// TIA Portal V20 export
FUNCTION_BLOCK "Sequence_1_SemiAutoSplice"   // FB124, LAD
TITLE = Sequence
// Sequence template programmend in ladder logic
// stored: IsIECCheckEnabled true, MemoryReserve 100, Namespace Unit1.Em2, SetENOAutomatically true
   VAR
      instSequenceLADControl { ExternalWritable := 'False'} : "LAF_ControlLadSequence";
      instSequenceLADStatus { ExternalWritable := 'False'} : "LAF_StatusLadSequence";
      statPulse { ExternalWritable := 'False'} : Array[0..999] of Bool;
      statTonTimer { ExternalWritable := 'False'} : Array[0..9999] of TON_TIME;
   END_VAR
   VAR_TEMP
      tempCustomerAction : Bool;   // Placeholder for possible actions
      tempDo_nothing_and_wait_for_init : Bool;   // Placeholder for doing nothing
      tempSafeStateCondition : Bool;   // Temp Condition for the equipment module to be in a safe state
   END_VAR
   VAR CONSTANT
      STEP_IDLE : DInt := 1;   // Idle Step
      JOB_1_STEP_01 : DInt := 101;   // Template Step
      JOB_1_STEP_11 : DInt := 111;   // Template Step
      JOB_2_STEP_01 : DInt := 201;   // Template Step
      JOB_2_STEP_11 : DInt := 211;   // Template Step
      JOB_2_STEP_21 : DInt := 221;   // Template Step
      JOB_2_STEP_31 : DInt := 231;   // Template Step
      JOB_2_STEP_41 : DInt := 241;   // Template Step
      JOB_3_STEP_01 : DInt := 301;   // Template Step
      JOB_3_STEP_03 : DInt := 303;
      JOB_3_STEP_11 : DInt := 311;
      JOB_3_STEP_21 : DInt := 321;
      JOB_3_STEP_31 : DInt := 331;
      JOB_3_STEP_41 : DInt := 341;
      JOB_3_STEP_51 : DInt := 351;
      JOB_4_STEP_01 : DInt := 401;   // Template Step
      JOB_4_STEP_03 : DInt := 403;   // Template Step
      JOB_4_STEP_11 : DInt := 411;   // Template Step
      JOB_4_STEP_21 : DInt := 421;   // Template Step
      JOB_4_STEP_31 : DInt := 431;   // Template Step
      JOB_4_STEP_41 : DInt := 441;
      JOB_4_STEP_51 : DInt := 451;
      JOB_5_STEP_01 : DInt := 501;   // Template Step
      JOB_6_STEP_01 : DInt := 601;   // Template Step
      JOB_7_STEP_01 : DInt := 701;   // Template Step
      JOB_7_STEP_11 : DInt := 711;   // Template Step
      JOB_7_STEP_21 : DInt := 721;   // Template Step
      JOB_7_STEP_31 : DInt := 731;   // Template Step
      JOB_8_STEP_01 : DInt := 801;   // Template Step
      JOB_8_STEP_11 : DInt := 811;   // Template Step
      JOB_9_STEP_01 : DInt := 901;   // Template Step
      JOB_9_STEP_11 : DInt := 911;   // Template Step
      JOB_9_STEP_21 : DInt := 921;   // Template Step
      JOB_10_STEP_01 : DInt := 1001;   // Template Step
      JOB_10_STEP_11 : DInt := 1011;   // Template Step
      JOB_10_STEP_21 : DInt := 1021;   // Template Step
      JOB_10_STEP_31 : DInt := 1031;   // Template Step
      JOB_10_STEP_41 : DInt := 1041;   // Template Step
      JOB_11_STEP_01 : DInt := 1101;   // Template Step
      JOB_11_STEP_11 : DInt := 1111;   // Template Step
      JOB_11_STEP_21 : DInt := 1121;   // Template Step
      JOB_12_STEP_01 : DInt := 1201;   // Template Step
      JOB_12_STEP_11 : DInt := 1211;   // Template Step
      JOB_12_STEP_21 : DInt := 1221;   // Template Step
      JOB_13_STEP_01 : DInt := 1301;   // Template Step
      JOB_13_STEP_11 : DInt := 1311;   // Template Step
      JOB_13_STEP_21 : DInt := 1321;   // Template Step
      JOB_13_STEP_31 : DInt := 1331;   // Template Step
      JOB_13_STEP_41 : DInt := 1341;   // Template Step
      JOB_13_STEP_45 : DInt := 1345;   // Template Step
      JOB_13_STEP_46 : DInt := 1346;   // Template Step
      JOB_13_STEP_48 : DInt := 1348;   // Template Step
      JOB_14_STEP_01 : DInt := 1401;   // Template Step
      JOB_14_STEP_11 : DInt := 1411;   // Template Step
      JOB_14_STEP_13 : DInt := 1413;   // Template Step
      JOB_14_STEP_21 : DInt := 1421;   // Template Step
      JOB_14_STEP_23 : DInt := 1423;   // Template Step
      JOB_14_STEP_31 : DInt := 1431;   // Template Step
      JOB_15_STEP_01 : DInt := 1501;   // Template Step
      JOB_15_STEP_11 : DInt := 1511;   // Template Step
      JOB_15_STEP_13 : DInt := 1513;   // Template Step
      JOB_15_STEP_21 : DInt := 1521;   // Template Step
      JOB_15_STEP_23 : DInt := 1523;   // Template Step
      JOB_15_STEP_31 : DInt := 1531;   // Template Step
      JOB_20_STEP_01 : DInt := 2001;   // Template Step
      JOB_20_STEP_04 : DInt := 2004;   // Template Step
      JOB_20_STEP_07 : DInt := 2007;   // Template Step
      JOB_20_STEP_10 : DInt := 2010;   // Template Step
      JOB_20_STEP_13 : DInt := 2013;   // Template Step
      JOB_20_STEP_16 : DInt := 2016;   // Template Step
      JOB_20_STEP_19 : DInt := 2019;   // Template Step
      JOB_20_STEP_22 : DInt := 2022;   // Template Step
      JOB_20_STEP_25 : DInt := 2025;   // Template Step
      JOB_20_STEP_28 : DInt := 2028;   // Template Step
      JOB_20_STEP_31 : DInt := 2031;   // Template Step
      JOB_20_STEP_34 : DInt := 2034;   // Template Step
      JOB_20_STEP_37 : DInt := 2037;   // Template Step
      JOB_20_STEP_40 : DInt := 2040;   // Template Step
      JOB_20_STEP_43 : DInt := 2043;   // Template Step
      JOB_20_STEP_46 : DInt := 2046;   // Template Step
      JOB_20_STEP_49 : DInt := 2049;   // Template Step
      JOB_20_STEP_52 : DInt := 2052;   // Template Step
      JOB_20_STEP_55 : DInt := 2055;   // Template Step
      JOB_20_STEP_58 : DInt := 2058;   // Template Step
      JOB_20_STEP_61 : DInt := 2061;   // Template Step
      JOB_20_STEP_64 : DInt := 2064;   // Template Step
      JOB_20_STEP_67 : DInt := 2067;   // Template Step
      JOB_20_STEP_70 : DInt := 2070;   // Template Step
      JOB_20_STEP_73 : DInt := 2073;   // Template Step
      JOB_20_STEP_76 : DInt := 2076;   // Template Step
      JOB_20_STEP_79 : DInt := 2079;   // Template Step
      JOB_20_STEP_82 : DInt := 2082;   // Template Step
      JOB_20_STEP_85 : DInt := 2085;   // Template Step
      JOB_20_STEP_88 : DInt := 2088;   // Template Step
      STEP_IMMEDIATE_STOP : DInt := 9001;   // Step executed when an immediate stop command is triggered for the sequence (i.e. when unit is in state aborting)
      TO_DO_INSERT_ACTIONS_HERE : Bool := TRUE;   // Template : Add actions
      TO_DO_INSERT_CONDITION_FOR_TRANSITION_HERE : Bool := TRUE;   // Template : Add conditions
      SeqDelayTime : Time := T#100ms;
      SeqNoDelayTime : Time;
      TRUE : Bool := TRUE;
      FALSE : Bool := FALSE;
   END_VAR
   VAR_TEMP   // added for the SCL form of the ladder/FBD networks
      _w1 : Bool;
      _w2 : Bool;
      _w3 : Bool;
   END_VAR
BEGIN

REGION Network 1: BLOCK INFO HEADER
   // (company) / (C) Copyright (year)
   // ---------------------------------------------------------------------------------
   // Title:                             (Title of this block)
   // Comment/Function: (that is implemented in the block)
   // Library/Family:           (that the source is dedicated to)
   // Author:                        (department / person in charge / contact)
   // Target System:          (test system with FW version)
   // Engineering:              TIA Portal (SW version)
   // Restrictions:               (OB types, etc.)
   // Requirements:           (hardware, technological package, etc.)
   // ---------------------------------------------------------------------------------
   // Change log table:
   // Version          | Date             | Signature      | Expert in charge  | Changes applied ------------------------|----------------------|-------------------------|--------------------------------|-----------------------
   // 001.000.000 | yyyy-mm-dd | 0x00000000 | (name of expert) | First released version
END_REGION

REGION Network 2: DESCRIPTION
   // This is a template block provided by the Automation Framework. It can be used to create an own project.
   // The Block Info Header is prepared to put in your own data.
   // Description of the block could be added here and the docu created by Code2Docu.
END_REGION

REGION Network 3: *************** CONTROL **********************
END_REGION

REGION Network 4: Sequence Control
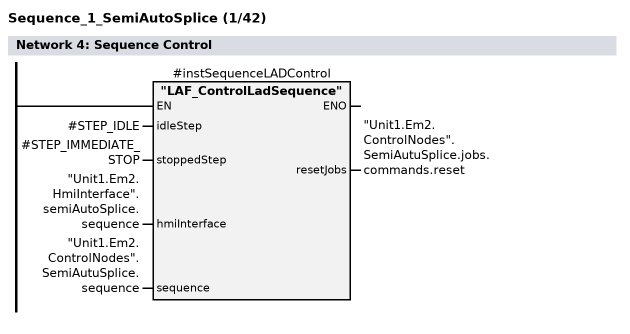
   RUNG wire#powerrail
      #instSequenceLADControl(idleStep := #STEP_IDLE, stoppedStep := #STEP_IMMEDIATE_STOP, hmiInterface := "Unit1.Em2.HmiInterface".semiAutoSplice.sequence, sequence := "Unit1.Em2.ControlNodes".SemiAutuSplice.sequence, resetJobs => "Unit1.Em2.ControlNodes".SemiAutuSplice.jobs.commands.reset)
   END_RUNG
   // the same network as SCL:
   #instSequenceLADControl(idleStep := #STEP_IDLE,   // "LAF_ControlLadSequence"
                           stoppedStep := #STEP_IMMEDIATE_STOP,
                           hmiInterface := "Unit1.Em2.HmiInterface".semiAutoSplice.sequence,
                           sequence := "Unit1.Em2.ControlNodes".SemiAutuSplice.sequence,
                           resetJobs => "Unit1.Em2.ControlNodes".SemiAutuSplice.jobs.commands.reset);
END_REGION

REGION Network 5: Step IDLE
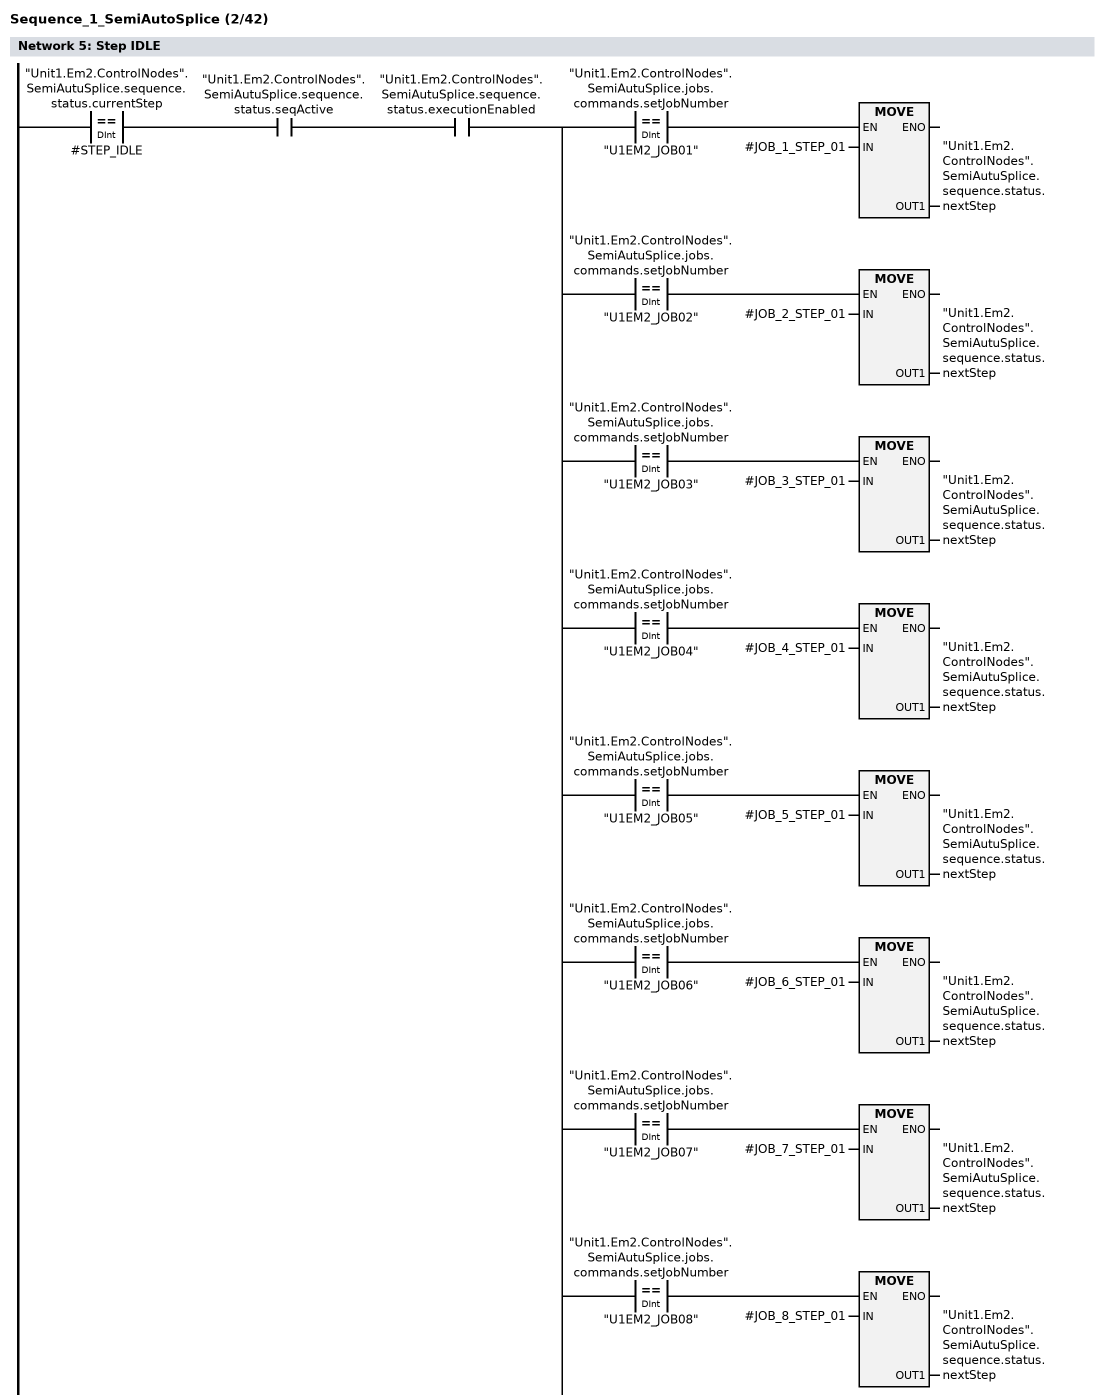
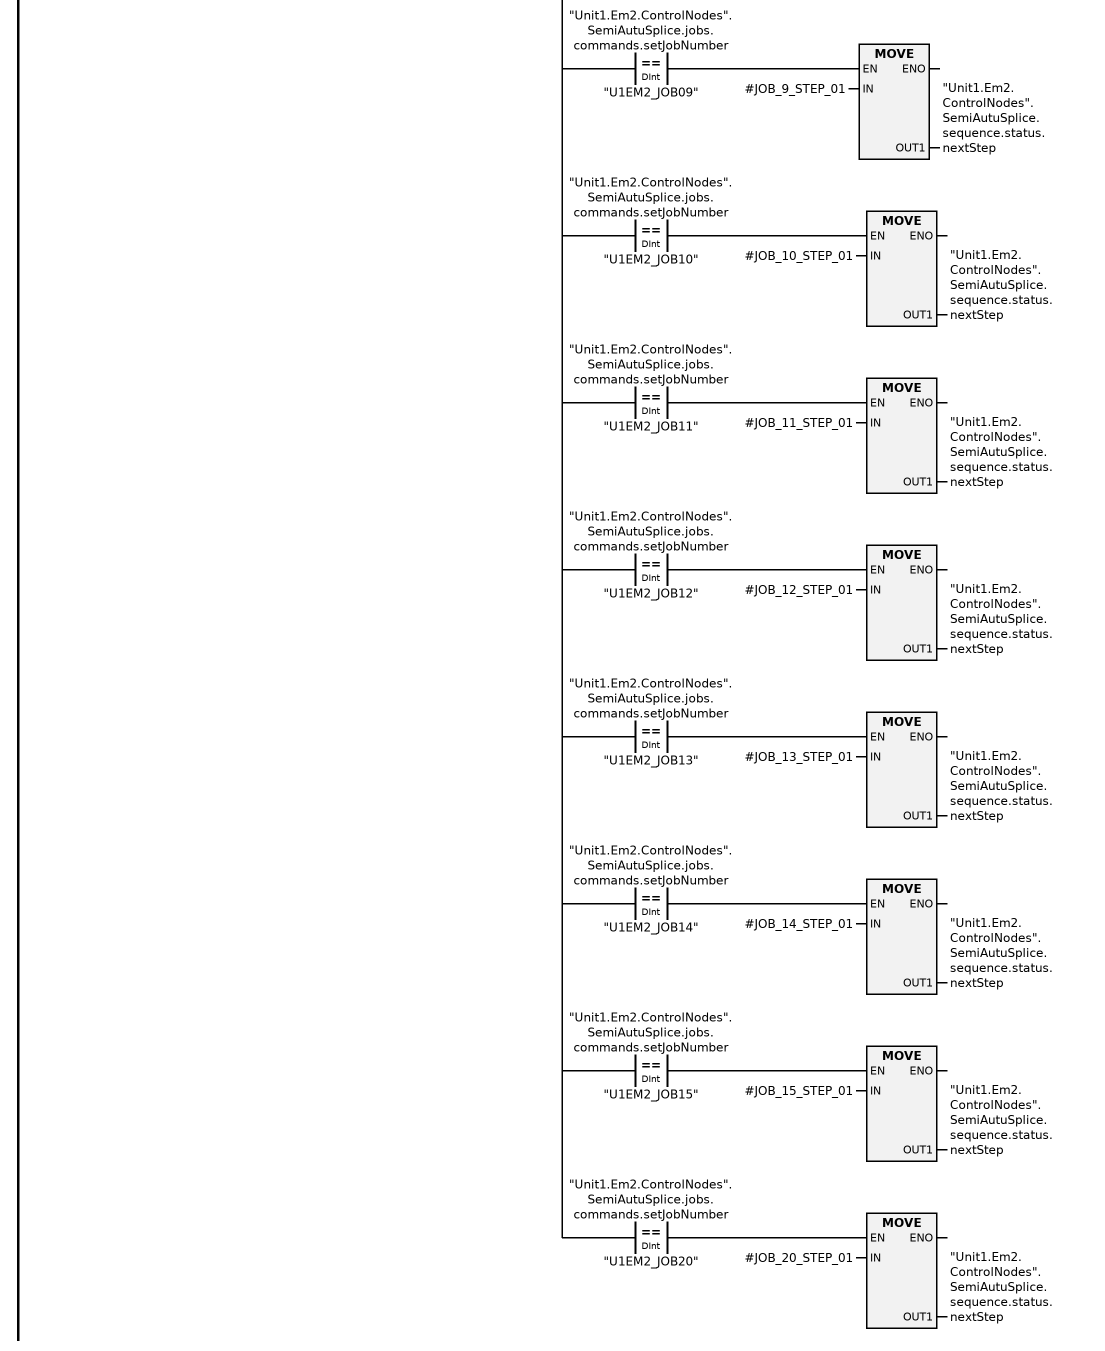
   RUNG wire#powerrail
      { S7_Templates := "SrcType := DInt" } EQ_Contact(in1 := "Unit1.Em2.ControlNodes".SemiAutuSplice.sequence.status.currentStep, in2 := #STEP_IDLE)
      Contact( "Unit1.Em2.ControlNodes".SemiAutuSplice.sequence.status.seqActive )
      Contact( "Unit1.Em2.ControlNodes".SemiAutuSplice.sequence.status.executionEnabled )
      wire#w1
      { S7_Templates := "SrcType := DInt" } EQ_Contact(in1 := "Unit1.Em2.ControlNodes".SemiAutuSplice.jobs.commands.setJobNumber, in2 := "U1EM2_JOB01")
      Move(in := #JOB_1_STEP_01, out1 => "Unit1.Em2.ControlNodes".SemiAutuSplice.sequence.status.nextStep)
   END_RUNG
   RUNG wire#w1
      { S7_Templates := "SrcType := DInt" } EQ_Contact(in1 := "Unit1.Em2.ControlNodes".SemiAutuSplice.jobs.commands.setJobNumber, in2 := "U1EM2_JOB02")
      Move(in := #JOB_2_STEP_01, out1 => "Unit1.Em2.ControlNodes".SemiAutuSplice.sequence.status.nextStep)
   END_RUNG
   RUNG wire#w1
      { S7_Templates := "SrcType := DInt" } EQ_Contact(in1 := "Unit1.Em2.ControlNodes".SemiAutuSplice.jobs.commands.setJobNumber, in2 := "U1EM2_JOB03")
      Move(in := #JOB_3_STEP_01, out1 => "Unit1.Em2.ControlNodes".SemiAutuSplice.sequence.status.nextStep)
   END_RUNG
   RUNG wire#w1
      { S7_Templates := "SrcType := DInt" } EQ_Contact(in1 := "Unit1.Em2.ControlNodes".SemiAutuSplice.jobs.commands.setJobNumber, in2 := "U1EM2_JOB04")
      Move(in := #JOB_4_STEP_01, out1 => "Unit1.Em2.ControlNodes".SemiAutuSplice.sequence.status.nextStep)
   END_RUNG
   RUNG wire#w1
      { S7_Templates := "SrcType := DInt" } EQ_Contact(in1 := "Unit1.Em2.ControlNodes".SemiAutuSplice.jobs.commands.setJobNumber, in2 := "U1EM2_JOB05")
      Move(in := #JOB_5_STEP_01, out1 => "Unit1.Em2.ControlNodes".SemiAutuSplice.sequence.status.nextStep)
   END_RUNG
   RUNG wire#w1
      { S7_Templates := "SrcType := DInt" } EQ_Contact(in1 := "Unit1.Em2.ControlNodes".SemiAutuSplice.jobs.commands.setJobNumber, in2 := "U1EM2_JOB06")
      Move(in := #JOB_6_STEP_01, out1 => "Unit1.Em2.ControlNodes".SemiAutuSplice.sequence.status.nextStep)
   END_RUNG
   RUNG wire#w1
      { S7_Templates := "SrcType := DInt" } EQ_Contact(in1 := "Unit1.Em2.ControlNodes".SemiAutuSplice.jobs.commands.setJobNumber, in2 := "U1EM2_JOB07")
      Move(in := #JOB_7_STEP_01, out1 => "Unit1.Em2.ControlNodes".SemiAutuSplice.sequence.status.nextStep)
   END_RUNG
   RUNG wire#w1
      { S7_Templates := "SrcType := DInt" } EQ_Contact(in1 := "Unit1.Em2.ControlNodes".SemiAutuSplice.jobs.commands.setJobNumber, in2 := "U1EM2_JOB08")
      Move(in := #JOB_8_STEP_01, out1 => "Unit1.Em2.ControlNodes".SemiAutuSplice.sequence.status.nextStep)
   END_RUNG
   RUNG wire#w1
      { S7_Templates := "SrcType := DInt" } EQ_Contact(in1 := "Unit1.Em2.ControlNodes".SemiAutuSplice.jobs.commands.setJobNumber, in2 := "U1EM2_JOB09")
      Move(in := #JOB_9_STEP_01, out1 => "Unit1.Em2.ControlNodes".SemiAutuSplice.sequence.status.nextStep)
   END_RUNG
   RUNG wire#w1
      { S7_Templates := "SrcType := DInt" } EQ_Contact(in1 := "Unit1.Em2.ControlNodes".SemiAutuSplice.jobs.commands.setJobNumber, in2 := "U1EM2_JOB10")
      Move(in := #JOB_10_STEP_01, out1 => "Unit1.Em2.ControlNodes".SemiAutuSplice.sequence.status.nextStep)
   END_RUNG
   RUNG wire#w1
      { S7_Templates := "SrcType := DInt" } EQ_Contact(in1 := "Unit1.Em2.ControlNodes".SemiAutuSplice.jobs.commands.setJobNumber, in2 := "U1EM2_JOB11")
      Move(in := #JOB_11_STEP_01, out1 => "Unit1.Em2.ControlNodes".SemiAutuSplice.sequence.status.nextStep)
   END_RUNG
   RUNG wire#w1
      { S7_Templates := "SrcType := DInt" } EQ_Contact(in1 := "Unit1.Em2.ControlNodes".SemiAutuSplice.jobs.commands.setJobNumber, in2 := "U1EM2_JOB12")
      Move(in := #JOB_12_STEP_01, out1 => "Unit1.Em2.ControlNodes".SemiAutuSplice.sequence.status.nextStep)
   END_RUNG
   RUNG wire#w1
      { S7_Templates := "SrcType := DInt" } EQ_Contact(in1 := "Unit1.Em2.ControlNodes".SemiAutuSplice.jobs.commands.setJobNumber, in2 := "U1EM2_JOB13")
      Move(in := #JOB_13_STEP_01, out1 => "Unit1.Em2.ControlNodes".SemiAutuSplice.sequence.status.nextStep)
   END_RUNG
   RUNG wire#w1
      { S7_Templates := "SrcType := DInt" } EQ_Contact(in1 := "Unit1.Em2.ControlNodes".SemiAutuSplice.jobs.commands.setJobNumber, in2 := "U1EM2_JOB14")
      Move(in := #JOB_14_STEP_01, out1 => "Unit1.Em2.ControlNodes".SemiAutuSplice.sequence.status.nextStep)
   END_RUNG
   RUNG wire#w1
      { S7_Templates := "SrcType := DInt" } EQ_Contact(in1 := "Unit1.Em2.ControlNodes".SemiAutuSplice.jobs.commands.setJobNumber, in2 := "U1EM2_JOB15")
      Move(in := #JOB_15_STEP_01, out1 => "Unit1.Em2.ControlNodes".SemiAutuSplice.sequence.status.nextStep)
   END_RUNG
   RUNG wire#w1
      { S7_Templates := "SrcType := DInt" } EQ_Contact(in1 := "Unit1.Em2.ControlNodes".SemiAutuSplice.jobs.commands.setJobNumber, in2 := "U1EM2_JOB20")
      Move(in := #JOB_20_STEP_01, out1 => "Unit1.Em2.ControlNodes".SemiAutuSplice.sequence.status.nextStep)
   END_RUNG
   // the same network as SCL:
   #_w1 := ("Unit1.Em2.ControlNodes".SemiAutuSplice.sequence.status.currentStep = #STEP_IDLE) AND "Unit1.Em2.ControlNodes".SemiAutuSplice.sequence.status.seqActive AND "Unit1.Em2.ControlNodes".SemiAutuSplice.sequence.status.executionEnabled;
   IF #_w1 AND ("Unit1.Em2.ControlNodes".SemiAutuSplice.jobs.commands.setJobNumber = "U1EM2_JOB01") THEN
       "Unit1.Em2.ControlNodes".SemiAutuSplice.sequence.status.nextStep := #JOB_1_STEP_01;
   END_IF;
   IF #_w1 AND ("Unit1.Em2.ControlNodes".SemiAutuSplice.jobs.commands.setJobNumber = "U1EM2_JOB02") THEN
       "Unit1.Em2.ControlNodes".SemiAutuSplice.sequence.status.nextStep := #JOB_2_STEP_01;
   END_IF;
   IF #_w1 AND ("Unit1.Em2.ControlNodes".SemiAutuSplice.jobs.commands.setJobNumber = "U1EM2_JOB03") THEN
       "Unit1.Em2.ControlNodes".SemiAutuSplice.sequence.status.nextStep := #JOB_3_STEP_01;
   END_IF;
   IF #_w1 AND ("Unit1.Em2.ControlNodes".SemiAutuSplice.jobs.commands.setJobNumber = "U1EM2_JOB04") THEN
       "Unit1.Em2.ControlNodes".SemiAutuSplice.sequence.status.nextStep := #JOB_4_STEP_01;
   END_IF;
   IF #_w1 AND ("Unit1.Em2.ControlNodes".SemiAutuSplice.jobs.commands.setJobNumber = "U1EM2_JOB05") THEN
       "Unit1.Em2.ControlNodes".SemiAutuSplice.sequence.status.nextStep := #JOB_5_STEP_01;
   END_IF;
   IF #_w1 AND ("Unit1.Em2.ControlNodes".SemiAutuSplice.jobs.commands.setJobNumber = "U1EM2_JOB06") THEN
       "Unit1.Em2.ControlNodes".SemiAutuSplice.sequence.status.nextStep := #JOB_6_STEP_01;
   END_IF;
   IF #_w1 AND ("Unit1.Em2.ControlNodes".SemiAutuSplice.jobs.commands.setJobNumber = "U1EM2_JOB07") THEN
       "Unit1.Em2.ControlNodes".SemiAutuSplice.sequence.status.nextStep := #JOB_7_STEP_01;
   END_IF;
   IF #_w1 AND ("Unit1.Em2.ControlNodes".SemiAutuSplice.jobs.commands.setJobNumber = "U1EM2_JOB08") THEN
       "Unit1.Em2.ControlNodes".SemiAutuSplice.sequence.status.nextStep := #JOB_8_STEP_01;
   END_IF;
   IF #_w1 AND ("Unit1.Em2.ControlNodes".SemiAutuSplice.jobs.commands.setJobNumber = "U1EM2_JOB09") THEN
       "Unit1.Em2.ControlNodes".SemiAutuSplice.sequence.status.nextStep := #JOB_9_STEP_01;
   END_IF;
   IF #_w1 AND ("Unit1.Em2.ControlNodes".SemiAutuSplice.jobs.commands.setJobNumber = "U1EM2_JOB10") THEN
       "Unit1.Em2.ControlNodes".SemiAutuSplice.sequence.status.nextStep := #JOB_10_STEP_01;
   END_IF;
   IF #_w1 AND ("Unit1.Em2.ControlNodes".SemiAutuSplice.jobs.commands.setJobNumber = "U1EM2_JOB11") THEN
       "Unit1.Em2.ControlNodes".SemiAutuSplice.sequence.status.nextStep := #JOB_11_STEP_01;
   END_IF;
   IF #_w1 AND ("Unit1.Em2.ControlNodes".SemiAutuSplice.jobs.commands.setJobNumber = "U1EM2_JOB12") THEN
       "Unit1.Em2.ControlNodes".SemiAutuSplice.sequence.status.nextStep := #JOB_12_STEP_01;
   END_IF;
   IF #_w1 AND ("Unit1.Em2.ControlNodes".SemiAutuSplice.jobs.commands.setJobNumber = "U1EM2_JOB13") THEN
       "Unit1.Em2.ControlNodes".SemiAutuSplice.sequence.status.nextStep := #JOB_13_STEP_01;
   END_IF;
   IF #_w1 AND ("Unit1.Em2.ControlNodes".SemiAutuSplice.jobs.commands.setJobNumber = "U1EM2_JOB14") THEN
       "Unit1.Em2.ControlNodes".SemiAutuSplice.sequence.status.nextStep := #JOB_14_STEP_01;
   END_IF;
   IF #_w1 AND ("Unit1.Em2.ControlNodes".SemiAutuSplice.jobs.commands.setJobNumber = "U1EM2_JOB15") THEN
       "Unit1.Em2.ControlNodes".SemiAutuSplice.sequence.status.nextStep := #JOB_15_STEP_01;
   END_IF;
   IF #_w1 AND ("Unit1.Em2.ControlNodes".SemiAutuSplice.jobs.commands.setJobNumber = "U1EM2_JOB20") THEN
       "Unit1.Em2.ControlNodes".SemiAutuSplice.sequence.status.nextStep := #JOB_20_STEP_01;
   END_IF;
END_REGION

REGION Network 6: Step IDLE Stopper WorkPos Command
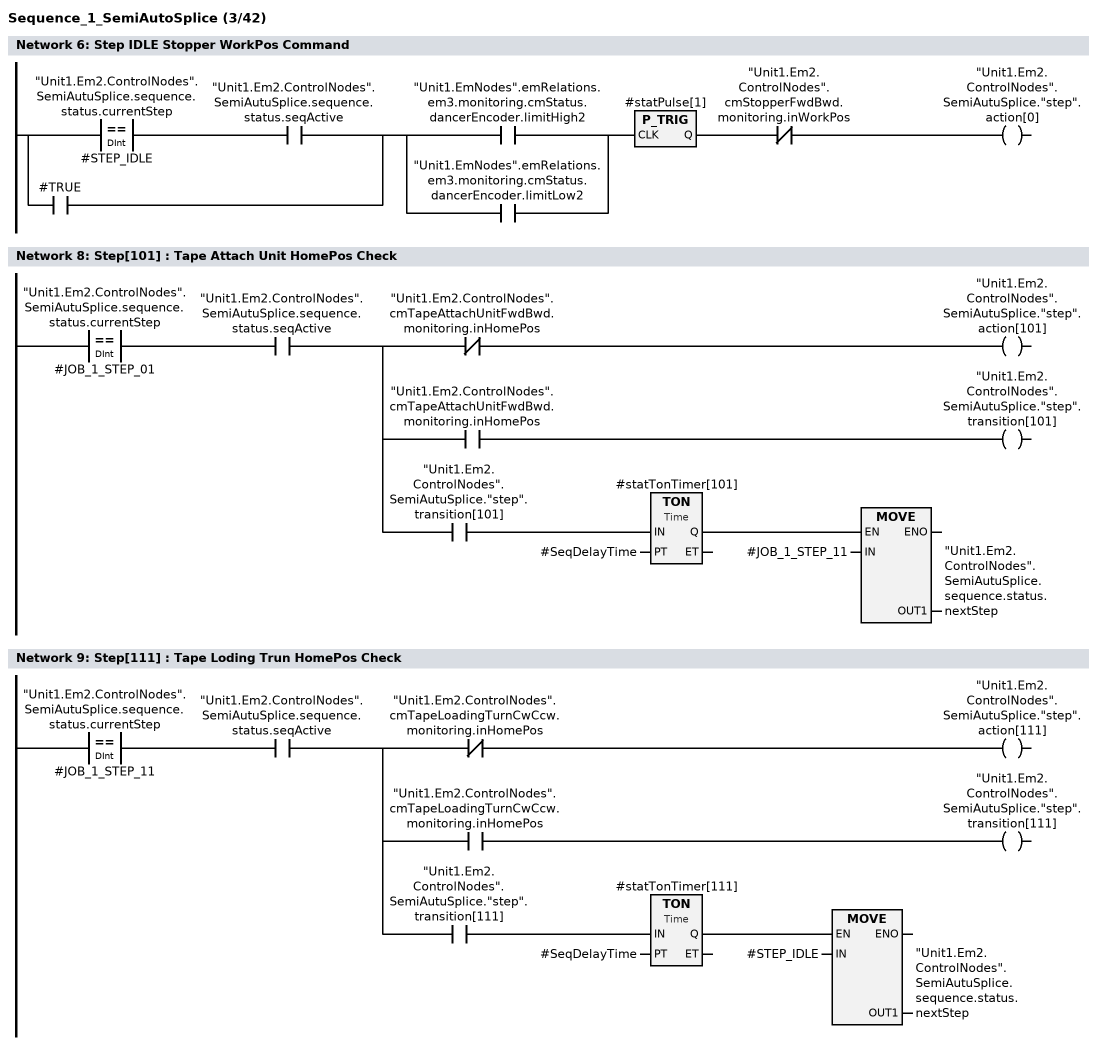
   RUNG wire#powerrail
      { S7_Templates := "SrcType := DInt" } EQ_Contact(in1 := "Unit1.Em2.ControlNodes".SemiAutuSplice.sequence.status.currentStep, in2 := #STEP_IDLE)
      Contact( "Unit1.Em2.ControlNodes".SemiAutuSplice.sequence.status.seqActive )
      wire#w1
      Contact( "Unit1.EmNodes".emRelations.em3.monitoring.cmStatus.dancerEncoder.limitHigh2 )
      wire#w2
      P_Trig( #statPulse[1] )
      I_Contact( "Unit1.Em2.ControlNodes".cmStopperFwdBwd.monitoring.inWorkPos )
      Coil( "Unit1.Em2.ControlNodes".SemiAutuSplice."step".action[0] )
   END_RUNG
   RUNG wire#powerrail
      Contact( #TRUE )
   END_RUNG wire#w1
   RUNG wire#w1
      Contact( "Unit1.EmNodes".emRelations.em3.monitoring.cmStatus.dancerEncoder.limitLow2 )
   END_RUNG wire#w2
   // the same network as SCL:
   #_w1 := ((("Unit1.Em2.ControlNodes".SemiAutuSplice.sequence.status.currentStep = #STEP_IDLE) AND "Unit1.Em2.ControlNodes".SemiAutuSplice.sequence.status.seqActive) OR #TRUE) AND ("Unit1.EmNodes".emRelations.em3.monitoring.cmStatus.dancerEncoder.limitHigh2 OR "Unit1.EmNodes".emRelations.em3.monitoring.cmStatus.dancerEncoder.limitLow2);
   #_w2 := #_w1 AND NOT #statPulse[1];   // rising edge
   #statPulse[1] := #_w1;
   "Unit1.Em2.ControlNodes".SemiAutuSplice."step".action[0] := #_w2 AND NOT "Unit1.Em2.ControlNodes".cmStopperFwdBwd.monitoring.inWorkPos;
END_REGION

REGION Network 7: ******************** JOB[1] TAPE UNIT INITIALIZED ********************
END_REGION

REGION Network 8: Step[101] : Tape Attach Unit HomePos Check
   RUNG wire#powerrail
      { S7_Templates := "SrcType := DInt" } EQ_Contact(in1 := "Unit1.Em2.ControlNodes".SemiAutuSplice.sequence.status.currentStep, in2 := #JOB_1_STEP_01)
      Contact( "Unit1.Em2.ControlNodes".SemiAutuSplice.sequence.status.seqActive )
      wire#w1
      I_Contact( "Unit1.Em2.ControlNodes".cmTapeAttachUnitFwdBwd.monitoring.inHomePos )
      Coil( "Unit1.Em2.ControlNodes".SemiAutuSplice."step".action[101] )
   END_RUNG
   RUNG wire#w1
      Contact( "Unit1.Em2.ControlNodes".cmTapeAttachUnitFwdBwd.monitoring.inHomePos )
      Coil( "Unit1.Em2.ControlNodes".SemiAutuSplice."step".transition[101] )
   END_RUNG
   RUNG wire#w1
      Contact( "Unit1.Em2.ControlNodes".SemiAutuSplice."step".transition[101] )
      { S7_Templates := "time_type := Time" } #statTonTimer[101].TON(pt := #SeqDelayTime, et =>)
      Move(in := #JOB_1_STEP_11, out1 => "Unit1.Em2.ControlNodes".SemiAutuSplice.sequence.status.nextStep)
   END_RUNG
   // the same network as SCL:
   #_w1 := ("Unit1.Em2.ControlNodes".SemiAutuSplice.sequence.status.currentStep = #JOB_1_STEP_01) AND "Unit1.Em2.ControlNodes".SemiAutuSplice.sequence.status.seqActive;
   "Unit1.Em2.ControlNodes".SemiAutuSplice."step".action[101] := #_w1 AND NOT "Unit1.Em2.ControlNodes".cmTapeAttachUnitFwdBwd.monitoring.inHomePos;
   "Unit1.Em2.ControlNodes".SemiAutuSplice."step".transition[101] := #_w1 AND "Unit1.Em2.ControlNodes".cmTapeAttachUnitFwdBwd.monitoring.inHomePos;
   #statTonTimer[101].TON(IN := #_w1 AND "Unit1.Em2.ControlNodes".SemiAutuSplice."step".transition[101],
                          PT := #SeqDelayTime);
   IF #statTonTimer[101].Q THEN
       "Unit1.Em2.ControlNodes".SemiAutuSplice.sequence.status.nextStep := #JOB_1_STEP_11;
   END_IF;
END_REGION

REGION Network 9: Step[111] : Tape Loding Trun HomePos Check
   RUNG wire#powerrail
      { S7_Templates := "SrcType := DInt" } EQ_Contact(in1 := "Unit1.Em2.ControlNodes".SemiAutuSplice.sequence.status.currentStep, in2 := #JOB_1_STEP_11)
      Contact( "Unit1.Em2.ControlNodes".SemiAutuSplice.sequence.status.seqActive )
      wire#w1
      I_Contact( "Unit1.Em2.ControlNodes".cmTapeLoadingTurnCwCcw.monitoring.inHomePos )
      Coil( "Unit1.Em2.ControlNodes".SemiAutuSplice."step".action[111] )
   END_RUNG
   RUNG wire#w1
      Contact( "Unit1.Em2.ControlNodes".cmTapeLoadingTurnCwCcw.monitoring.inHomePos )
      Coil( "Unit1.Em2.ControlNodes".SemiAutuSplice."step".transition[111] )
   END_RUNG
   RUNG wire#w1
      Contact( "Unit1.Em2.ControlNodes".SemiAutuSplice."step".transition[111] )
      { S7_Templates := "time_type := Time" } #statTonTimer[111].TON(pt := #SeqDelayTime, et =>)
      Move(in := #STEP_IDLE, out1 => "Unit1.Em2.ControlNodes".SemiAutuSplice.sequence.status.nextStep)
   END_RUNG
   // the same network as SCL:
   #_w1 := ("Unit1.Em2.ControlNodes".SemiAutuSplice.sequence.status.currentStep = #JOB_1_STEP_11) AND "Unit1.Em2.ControlNodes".SemiAutuSplice.sequence.status.seqActive;
   "Unit1.Em2.ControlNodes".SemiAutuSplice."step".action[111] := #_w1 AND NOT "Unit1.Em2.ControlNodes".cmTapeLoadingTurnCwCcw.monitoring.inHomePos;
   "Unit1.Em2.ControlNodes".SemiAutuSplice."step".transition[111] := #_w1 AND "Unit1.Em2.ControlNodes".cmTapeLoadingTurnCwCcw.monitoring.inHomePos;
   #statTonTimer[111].TON(IN := #_w1 AND "Unit1.Em2.ControlNodes".SemiAutuSplice."step".transition[111],
                          PT := #SeqDelayTime);
   IF #statTonTimer[111].Q THEN
       "Unit1.Em2.ControlNodes".SemiAutuSplice.sequence.status.nextStep := #STEP_IDLE;
   END_IF;
END_REGION

REGION Network 10: ******************** JOB[2] AUTO SPLICER MODULE INITIALIZED ********************
END_REGION

REGION Network 11: Step[201] : Uw Semi Splicer Vacuum ALL HomePos Check
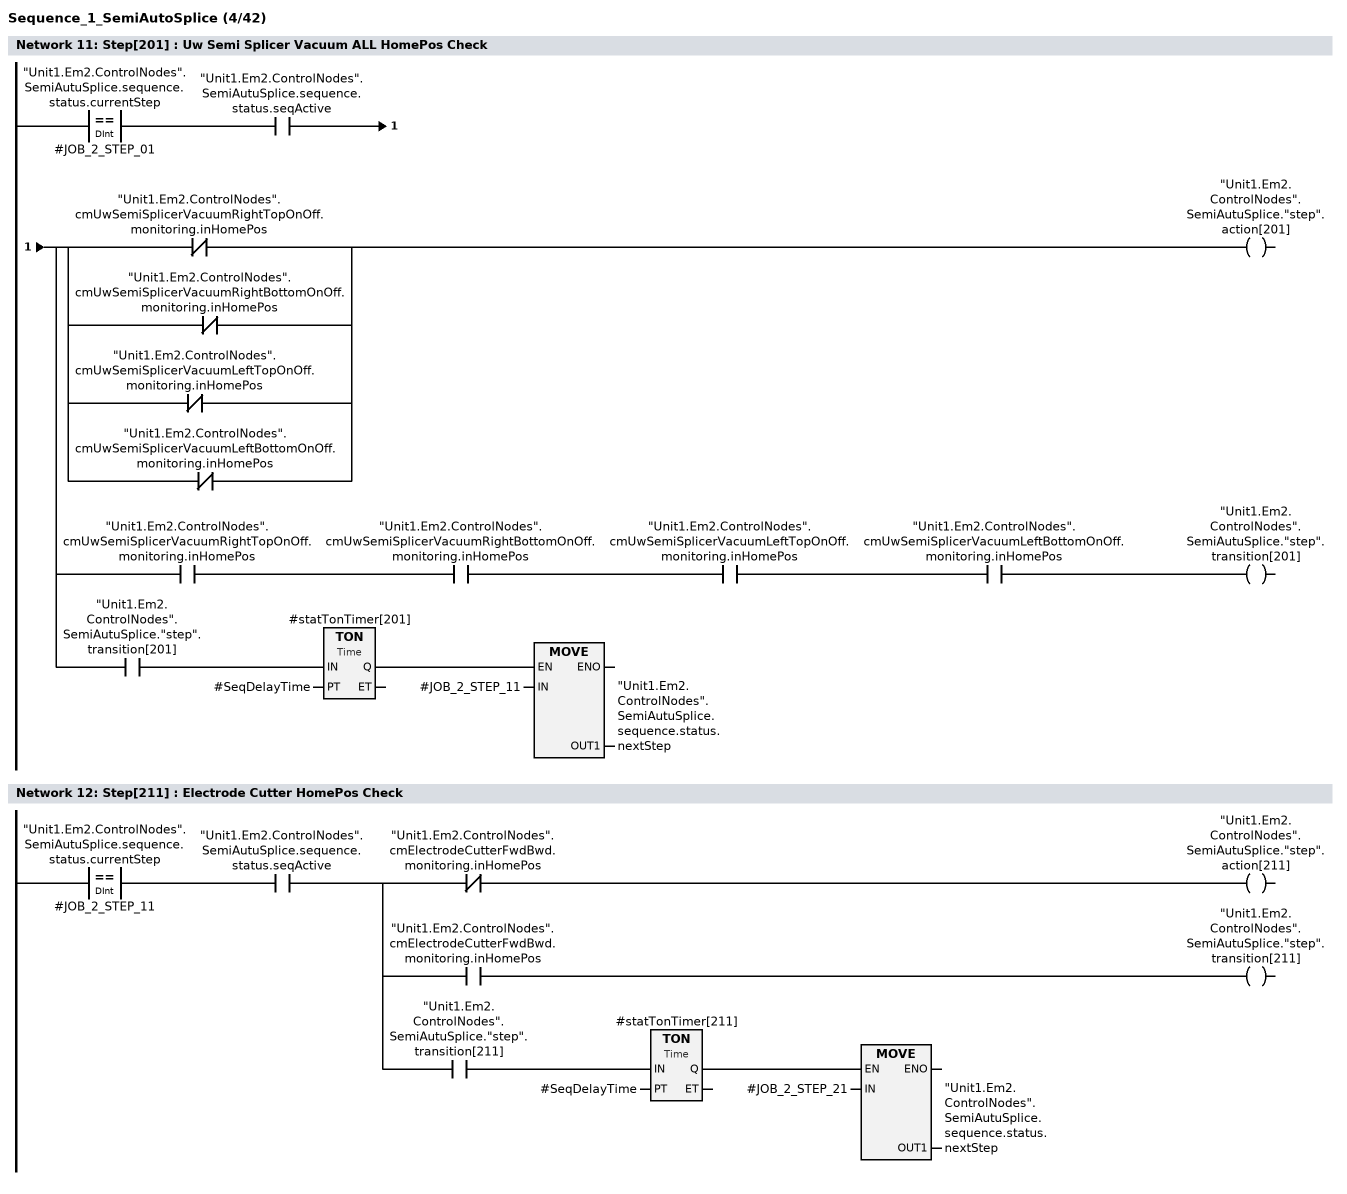
   RUNG wire#powerrail
      { S7_Templates := "SrcType := DInt" } EQ_Contact(in1 := "Unit1.Em2.ControlNodes".SemiAutuSplice.sequence.status.currentStep, in2 := #JOB_2_STEP_01)
      Contact( "Unit1.Em2.ControlNodes".SemiAutuSplice.sequence.status.seqActive )
      wire#w1
      I_Contact( "Unit1.Em2.ControlNodes".cmUwSemiSplicerVacuumRightTopOnOff.monitoring.inHomePos )
      wire#w2
      Coil( "Unit1.Em2.ControlNodes".SemiAutuSplice."step".action[201] )
   END_RUNG
   RUNG wire#w1
      I_Contact( "Unit1.Em2.ControlNodes".cmUwSemiSplicerVacuumRightBottomOnOff.monitoring.inHomePos )
   END_RUNG wire#w2
   RUNG wire#w1
      I_Contact( "Unit1.Em2.ControlNodes".cmUwSemiSplicerVacuumLeftTopOnOff.monitoring.inHomePos )
   END_RUNG wire#w2
   RUNG wire#w1
      I_Contact( "Unit1.Em2.ControlNodes".cmUwSemiSplicerVacuumLeftBottomOnOff.monitoring.inHomePos )
   END_RUNG wire#w2
   RUNG wire#w1
      Contact( "Unit1.Em2.ControlNodes".cmUwSemiSplicerVacuumRightTopOnOff.monitoring.inHomePos )
      Contact( "Unit1.Em2.ControlNodes".cmUwSemiSplicerVacuumRightBottomOnOff.monitoring.inHomePos )
      Contact( "Unit1.Em2.ControlNodes".cmUwSemiSplicerVacuumLeftTopOnOff.monitoring.inHomePos )
      Contact( "Unit1.Em2.ControlNodes".cmUwSemiSplicerVacuumLeftBottomOnOff.monitoring.inHomePos )
      Coil( "Unit1.Em2.ControlNodes".SemiAutuSplice."step".transition[201] )
   END_RUNG
   RUNG wire#w1
      Contact( "Unit1.Em2.ControlNodes".SemiAutuSplice."step".transition[201] )
      { S7_Templates := "time_type := Time" } #statTonTimer[201].TON(pt := #SeqDelayTime, et =>)
      Move(in := #JOB_2_STEP_11, out1 => "Unit1.Em2.ControlNodes".SemiAutuSplice.sequence.status.nextStep)
   END_RUNG
   // the same network as SCL:
   #_w1 := ("Unit1.Em2.ControlNodes".SemiAutuSplice.sequence.status.currentStep = #JOB_2_STEP_01) AND "Unit1.Em2.ControlNodes".SemiAutuSplice.sequence.status.seqActive;
   "Unit1.Em2.ControlNodes".SemiAutuSplice."step".action[201] := #_w1 AND (NOT "Unit1.Em2.ControlNodes".cmUwSemiSplicerVacuumRightTopOnOff.monitoring.inHomePos OR NOT "Unit1.Em2.ControlNodes".cmUwSemiSplicerVacuumRightBottomOnOff.monitoring.inHomePos OR NOT "Unit1.Em2.ControlNodes".cmUwSemiSplicerVacuumLeftTopOnOff.monitoring.inHomePos OR NOT "Unit1.Em2.ControlNodes".cmUwSemiSplicerVacuumLeftBottomOnOff.monitoring.inHomePos);
   "Unit1.Em2.ControlNodes".SemiAutuSplice."step".transition[201] := #_w1 AND "Unit1.Em2.ControlNodes".cmUwSemiSplicerVacuumRightTopOnOff.monitoring.inHomePos AND "Unit1.Em2.ControlNodes".cmUwSemiSplicerVacuumRightBottomOnOff.monitoring.inHomePos AND "Unit1.Em2.ControlNodes".cmUwSemiSplicerVacuumLeftTopOnOff.monitoring.inHomePos AND "Unit1.Em2.ControlNodes".cmUwSemiSplicerVacuumLeftBottomOnOff.monitoring.inHomePos;
   #statTonTimer[201].TON(IN := #_w1 AND "Unit1.Em2.ControlNodes".SemiAutuSplice."step".transition[201],
                          PT := #SeqDelayTime);
   IF #statTonTimer[201].Q THEN
       "Unit1.Em2.ControlNodes".SemiAutuSplice.sequence.status.nextStep := #JOB_2_STEP_11;
   END_IF;
END_REGION

REGION Network 12: Step[211] : Electrode Cutter HomePos Check
   RUNG wire#powerrail
      { S7_Templates := "SrcType := DInt" } EQ_Contact(in1 := "Unit1.Em2.ControlNodes".SemiAutuSplice.sequence.status.currentStep, in2 := #JOB_2_STEP_11)
      Contact( "Unit1.Em2.ControlNodes".SemiAutuSplice.sequence.status.seqActive )
      wire#w1
      I_Contact( "Unit1.Em2.ControlNodes".cmElectrodeCutterFwdBwd.monitoring.inHomePos )
      Coil( "Unit1.Em2.ControlNodes".SemiAutuSplice."step".action[211] )
   END_RUNG
   RUNG wire#w1
      Contact( "Unit1.Em2.ControlNodes".cmElectrodeCutterFwdBwd.monitoring.inHomePos )
      Coil( "Unit1.Em2.ControlNodes".SemiAutuSplice."step".transition[211] )
   END_RUNG
   RUNG wire#w1
      Contact( "Unit1.Em2.ControlNodes".SemiAutuSplice."step".transition[211] )
      { S7_Templates := "time_type := Time" } #statTonTimer[211].TON(pt := #SeqDelayTime, et =>)
      Move(in := #JOB_2_STEP_21, out1 => "Unit1.Em2.ControlNodes".SemiAutuSplice.sequence.status.nextStep)
   END_RUNG
   // the same network as SCL:
   #_w1 := ("Unit1.Em2.ControlNodes".SemiAutuSplice.sequence.status.currentStep = #JOB_2_STEP_11) AND "Unit1.Em2.ControlNodes".SemiAutuSplice.sequence.status.seqActive;
   "Unit1.Em2.ControlNodes".SemiAutuSplice."step".action[211] := #_w1 AND NOT "Unit1.Em2.ControlNodes".cmElectrodeCutterFwdBwd.monitoring.inHomePos;
   "Unit1.Em2.ControlNodes".SemiAutuSplice."step".transition[211] := #_w1 AND "Unit1.Em2.ControlNodes".cmElectrodeCutterFwdBwd.monitoring.inHomePos;
   #statTonTimer[211].TON(IN := #_w1 AND "Unit1.Em2.ControlNodes".SemiAutuSplice."step".transition[211],
                          PT := #SeqDelayTime);
   IF #statTonTimer[211].Q THEN
       "Unit1.Em2.ControlNodes".SemiAutuSplice.sequence.status.nextStep := #JOB_2_STEP_21;
   END_IF;
END_REGION

REGION Network 13: Step[221] : Electrode Fix ALL HomePos Check
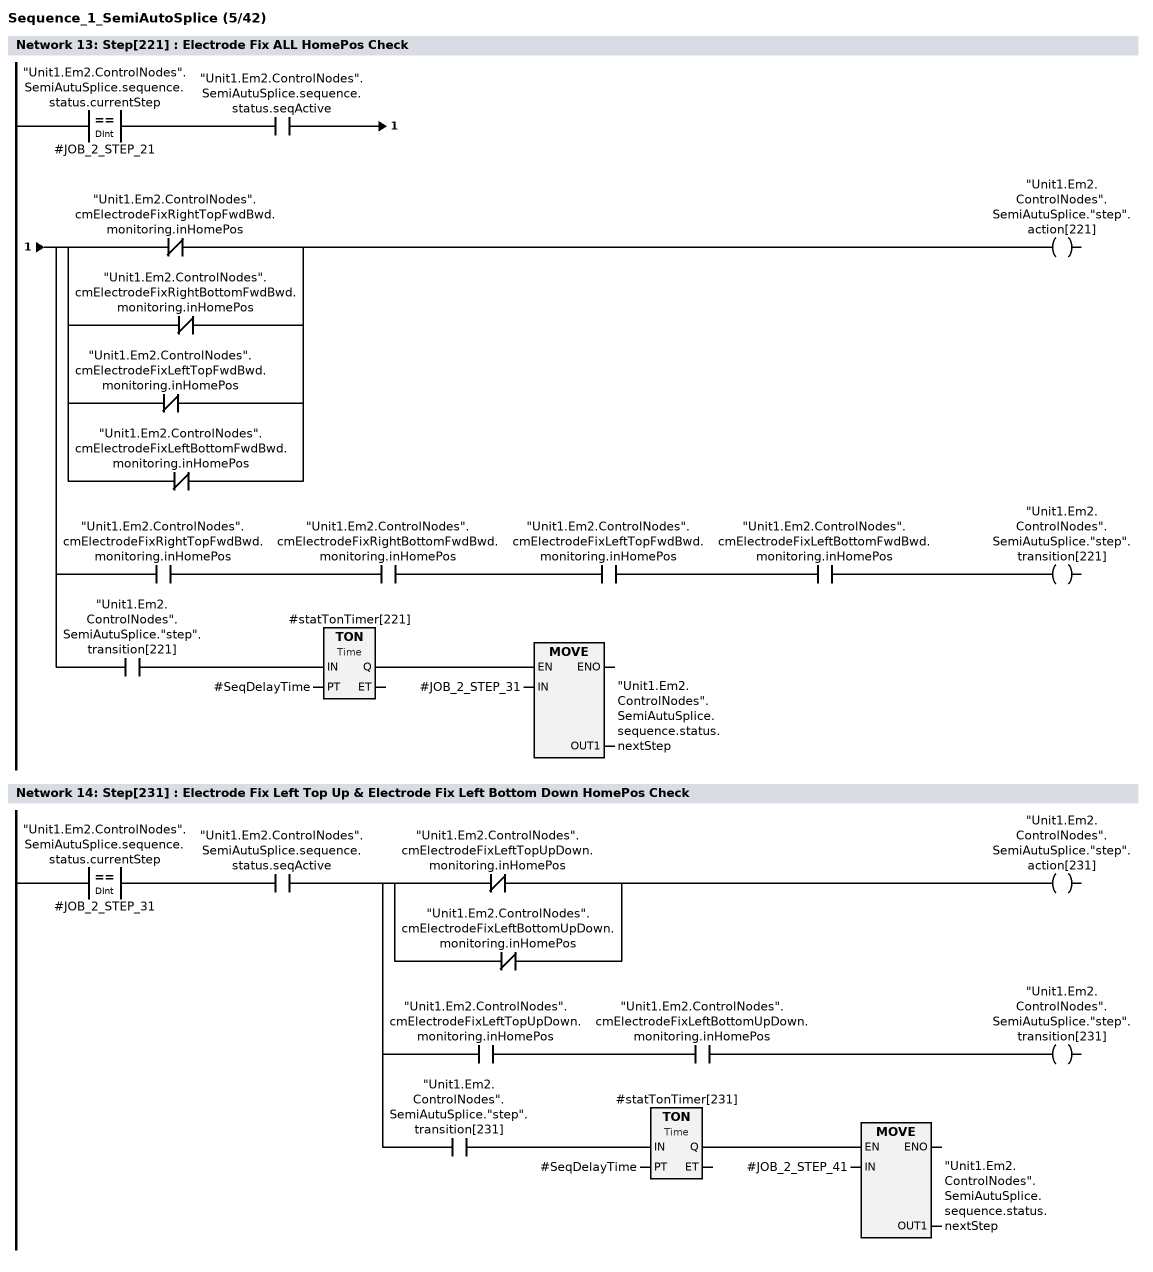
   RUNG wire#powerrail
      { S7_Templates := "SrcType := DInt" } EQ_Contact(in1 := "Unit1.Em2.ControlNodes".SemiAutuSplice.sequence.status.currentStep, in2 := #JOB_2_STEP_21)
      Contact( "Unit1.Em2.ControlNodes".SemiAutuSplice.sequence.status.seqActive )
      wire#w1
      I_Contact( "Unit1.Em2.ControlNodes".cmElectrodeFixRightTopFwdBwd.monitoring.inHomePos )
      wire#w2
      Coil( "Unit1.Em2.ControlNodes".SemiAutuSplice."step".action[221] )
   END_RUNG
   RUNG wire#w1
      I_Contact( "Unit1.Em2.ControlNodes".cmElectrodeFixRightBottomFwdBwd.monitoring.inHomePos )
   END_RUNG wire#w2
   RUNG wire#w1
      I_Contact( "Unit1.Em2.ControlNodes".cmElectrodeFixLeftTopFwdBwd.monitoring.inHomePos )
   END_RUNG wire#w2
   RUNG wire#w1
      I_Contact( "Unit1.Em2.ControlNodes".cmElectrodeFixLeftBottomFwdBwd.monitoring.inHomePos )
   END_RUNG wire#w2
   RUNG wire#w1
      Contact( "Unit1.Em2.ControlNodes".cmElectrodeFixRightTopFwdBwd.monitoring.inHomePos )
      Contact( "Unit1.Em2.ControlNodes".cmElectrodeFixRightBottomFwdBwd.monitoring.inHomePos )
      Contact( "Unit1.Em2.ControlNodes".cmElectrodeFixLeftTopFwdBwd.monitoring.inHomePos )
      Contact( "Unit1.Em2.ControlNodes".cmElectrodeFixLeftBottomFwdBwd.monitoring.inHomePos )
      Coil( "Unit1.Em2.ControlNodes".SemiAutuSplice."step".transition[221] )
   END_RUNG
   RUNG wire#w1
      Contact( "Unit1.Em2.ControlNodes".SemiAutuSplice."step".transition[221] )
      { S7_Templates := "time_type := Time" } #statTonTimer[221].TON(pt := #SeqDelayTime, et =>)
      Move(in := #JOB_2_STEP_31, out1 => "Unit1.Em2.ControlNodes".SemiAutuSplice.sequence.status.nextStep)
   END_RUNG
   // the same network as SCL:
   #_w1 := ("Unit1.Em2.ControlNodes".SemiAutuSplice.sequence.status.currentStep = #JOB_2_STEP_21) AND "Unit1.Em2.ControlNodes".SemiAutuSplice.sequence.status.seqActive;
   "Unit1.Em2.ControlNodes".SemiAutuSplice."step".action[221] := #_w1 AND (NOT "Unit1.Em2.ControlNodes".cmElectrodeFixRightTopFwdBwd.monitoring.inHomePos OR NOT "Unit1.Em2.ControlNodes".cmElectrodeFixRightBottomFwdBwd.monitoring.inHomePos OR NOT "Unit1.Em2.ControlNodes".cmElectrodeFixLeftTopFwdBwd.monitoring.inHomePos OR NOT "Unit1.Em2.ControlNodes".cmElectrodeFixLeftBottomFwdBwd.monitoring.inHomePos);
   "Unit1.Em2.ControlNodes".SemiAutuSplice."step".transition[221] := #_w1 AND "Unit1.Em2.ControlNodes".cmElectrodeFixRightTopFwdBwd.monitoring.inHomePos AND "Unit1.Em2.ControlNodes".cmElectrodeFixRightBottomFwdBwd.monitoring.inHomePos AND "Unit1.Em2.ControlNodes".cmElectrodeFixLeftTopFwdBwd.monitoring.inHomePos AND "Unit1.Em2.ControlNodes".cmElectrodeFixLeftBottomFwdBwd.monitoring.inHomePos;
   #statTonTimer[221].TON(IN := #_w1 AND "Unit1.Em2.ControlNodes".SemiAutuSplice."step".transition[221],
                          PT := #SeqDelayTime);
   IF #statTonTimer[221].Q THEN
       "Unit1.Em2.ControlNodes".SemiAutuSplice.sequence.status.nextStep := #JOB_2_STEP_31;
   END_IF;
END_REGION

REGION Network 14: Step[231] : Electrode Fix Left Top Up & Electrode Fix Left Bottom Down HomePos Check
   RUNG wire#powerrail
      { S7_Templates := "SrcType := DInt" } EQ_Contact(in1 := "Unit1.Em2.ControlNodes".SemiAutuSplice.sequence.status.currentStep, in2 := #JOB_2_STEP_31)
      Contact( "Unit1.Em2.ControlNodes".SemiAutuSplice.sequence.status.seqActive )
      wire#w1
      I_Contact( "Unit1.Em2.ControlNodes".cmElectrodeFixLeftTopUpDown.monitoring.inHomePos )
      wire#w2
      Coil( "Unit1.Em2.ControlNodes".SemiAutuSplice."step".action[231] )
   END_RUNG
   RUNG wire#w1
      I_Contact( "Unit1.Em2.ControlNodes".cmElectrodeFixLeftBottomUpDown.monitoring.inHomePos )
   END_RUNG wire#w2
   RUNG wire#w1
      Contact( "Unit1.Em2.ControlNodes".cmElectrodeFixLeftTopUpDown.monitoring.inHomePos )
      Contact( "Unit1.Em2.ControlNodes".cmElectrodeFixLeftBottomUpDown.monitoring.inHomePos )
      Coil( "Unit1.Em2.ControlNodes".SemiAutuSplice."step".transition[231] )
   END_RUNG
   RUNG wire#w1
      Contact( "Unit1.Em2.ControlNodes".SemiAutuSplice."step".transition[231] )
      { S7_Templates := "time_type := Time" } #statTonTimer[231].TON(pt := #SeqDelayTime, et =>)
      Move(in := #JOB_2_STEP_41, out1 => "Unit1.Em2.ControlNodes".SemiAutuSplice.sequence.status.nextStep)
   END_RUNG
   // the same network as SCL:
   #_w1 := ("Unit1.Em2.ControlNodes".SemiAutuSplice.sequence.status.currentStep = #JOB_2_STEP_31) AND "Unit1.Em2.ControlNodes".SemiAutuSplice.sequence.status.seqActive;
   "Unit1.Em2.ControlNodes".SemiAutuSplice."step".action[231] := #_w1 AND (NOT "Unit1.Em2.ControlNodes".cmElectrodeFixLeftTopUpDown.monitoring.inHomePos OR NOT "Unit1.Em2.ControlNodes".cmElectrodeFixLeftBottomUpDown.monitoring.inHomePos);
   "Unit1.Em2.ControlNodes".SemiAutuSplice."step".transition[231] := #_w1 AND "Unit1.Em2.ControlNodes".cmElectrodeFixLeftTopUpDown.monitoring.inHomePos AND "Unit1.Em2.ControlNodes".cmElectrodeFixLeftBottomUpDown.monitoring.inHomePos;
   #statTonTimer[231].TON(IN := #_w1 AND "Unit1.Em2.ControlNodes".SemiAutuSplice."step".transition[231],
                          PT := #SeqDelayTime);
   IF #statTonTimer[231].Q THEN
       "Unit1.Em2.ControlNodes".SemiAutuSplice.sequence.status.nextStep := #JOB_2_STEP_41;
   END_IF;
END_REGION

REGION Network 15: Step[241] : Stopper HomePos Check
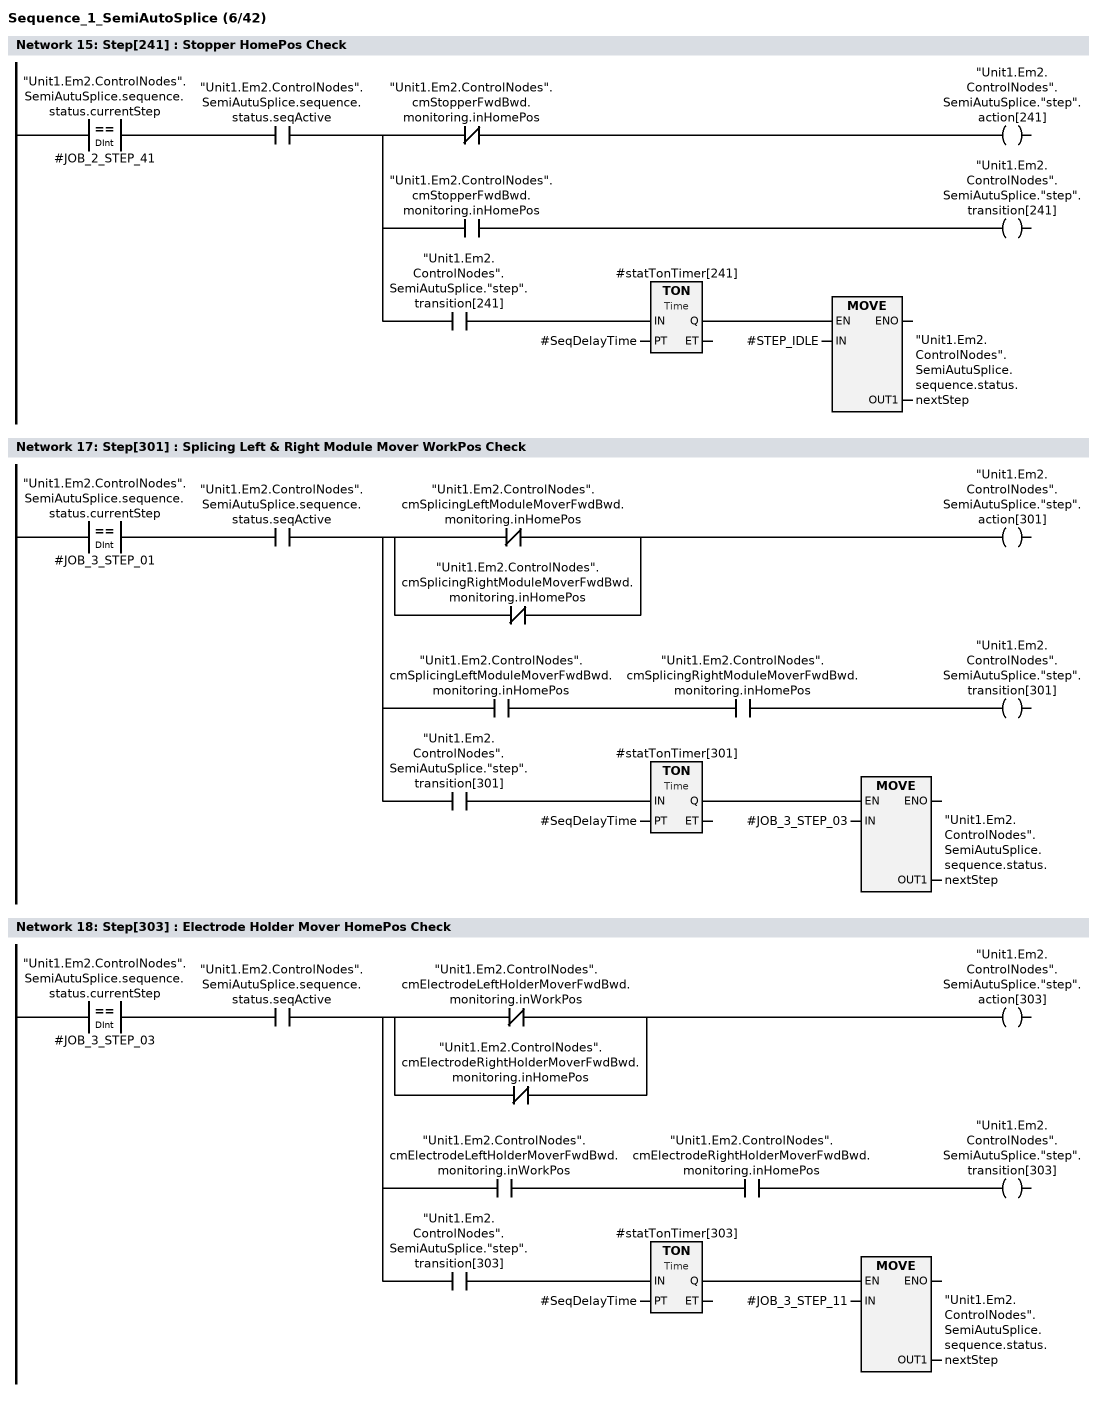
   RUNG wire#powerrail
      { S7_Templates := "SrcType := DInt" } EQ_Contact(in1 := "Unit1.Em2.ControlNodes".SemiAutuSplice.sequence.status.currentStep, in2 := #JOB_2_STEP_41)
      Contact( "Unit1.Em2.ControlNodes".SemiAutuSplice.sequence.status.seqActive )
      wire#w1
      I_Contact( "Unit1.Em2.ControlNodes".cmStopperFwdBwd.monitoring.inHomePos )
      Coil( "Unit1.Em2.ControlNodes".SemiAutuSplice."step".action[241] )
   END_RUNG
   RUNG wire#w1
      Contact( "Unit1.Em2.ControlNodes".cmStopperFwdBwd.monitoring.inHomePos )
      Coil( "Unit1.Em2.ControlNodes".SemiAutuSplice."step".transition[241] )
   END_RUNG
   RUNG wire#w1
      Contact( "Unit1.Em2.ControlNodes".SemiAutuSplice."step".transition[241] )
      { S7_Templates := "time_type := Time" } #statTonTimer[241].TON(pt := #SeqDelayTime, et =>)
      Move(in := #STEP_IDLE, out1 => "Unit1.Em2.ControlNodes".SemiAutuSplice.sequence.status.nextStep)
   END_RUNG
   // the same network as SCL:
   #_w1 := ("Unit1.Em2.ControlNodes".SemiAutuSplice.sequence.status.currentStep = #JOB_2_STEP_41) AND "Unit1.Em2.ControlNodes".SemiAutuSplice.sequence.status.seqActive;
   "Unit1.Em2.ControlNodes".SemiAutuSplice."step".action[241] := #_w1 AND NOT "Unit1.Em2.ControlNodes".cmStopperFwdBwd.monitoring.inHomePos;
   "Unit1.Em2.ControlNodes".SemiAutuSplice."step".transition[241] := #_w1 AND "Unit1.Em2.ControlNodes".cmStopperFwdBwd.monitoring.inHomePos;
   #statTonTimer[241].TON(IN := #_w1 AND "Unit1.Em2.ControlNodes".SemiAutuSplice."step".transition[241],
                          PT := #SeqDelayTime);
   IF #statTonTimer[241].Q THEN
       "Unit1.Em2.ControlNodes".SemiAutuSplice.sequence.status.nextStep := #STEP_IDLE;
   END_IF;
END_REGION

REGION Network 16: ******************** JOB[3] LEFT SPLICING MODULE MOVER INITIALIZED ********************
END_REGION

REGION Network 17: Step[301] : Splicing Left & Right Module Mover WorkPos Check
   RUNG wire#powerrail
      { S7_Templates := "SrcType := DInt" } EQ_Contact(in1 := "Unit1.Em2.ControlNodes".SemiAutuSplice.sequence.status.currentStep, in2 := #JOB_3_STEP_01)
      Contact( "Unit1.Em2.ControlNodes".SemiAutuSplice.sequence.status.seqActive )
      wire#w1
      I_Contact( "Unit1.Em2.ControlNodes".cmSplicingLeftModuleMoverFwdBwd.monitoring.inHomePos )
      wire#w2
      Coil( "Unit1.Em2.ControlNodes".SemiAutuSplice."step".action[301] )
   END_RUNG
   RUNG wire#w1
      I_Contact( "Unit1.Em2.ControlNodes".cmSplicingRightModuleMoverFwdBwd.monitoring.inHomePos )
   END_RUNG wire#w2
   RUNG wire#w1
      Contact( "Unit1.Em2.ControlNodes".cmSplicingLeftModuleMoverFwdBwd.monitoring.inHomePos )
      Contact( "Unit1.Em2.ControlNodes".cmSplicingRightModuleMoverFwdBwd.monitoring.inHomePos )
      Coil( "Unit1.Em2.ControlNodes".SemiAutuSplice."step".transition[301] )
   END_RUNG
   RUNG wire#w1
      Contact( "Unit1.Em2.ControlNodes".SemiAutuSplice."step".transition[301] )
      { S7_Templates := "time_type := Time" } #statTonTimer[301].TON(pt := #SeqDelayTime, et =>)
      Move(in := #JOB_3_STEP_03, out1 => "Unit1.Em2.ControlNodes".SemiAutuSplice.sequence.status.nextStep)
   END_RUNG
   // the same network as SCL:
   #_w1 := ("Unit1.Em2.ControlNodes".SemiAutuSplice.sequence.status.currentStep = #JOB_3_STEP_01) AND "Unit1.Em2.ControlNodes".SemiAutuSplice.sequence.status.seqActive;
   "Unit1.Em2.ControlNodes".SemiAutuSplice."step".action[301] := #_w1 AND (NOT "Unit1.Em2.ControlNodes".cmSplicingLeftModuleMoverFwdBwd.monitoring.inHomePos OR NOT "Unit1.Em2.ControlNodes".cmSplicingRightModuleMoverFwdBwd.monitoring.inHomePos);
   "Unit1.Em2.ControlNodes".SemiAutuSplice."step".transition[301] := #_w1 AND "Unit1.Em2.ControlNodes".cmSplicingLeftModuleMoverFwdBwd.monitoring.inHomePos AND "Unit1.Em2.ControlNodes".cmSplicingRightModuleMoverFwdBwd.monitoring.inHomePos;
   #statTonTimer[301].TON(IN := #_w1 AND "Unit1.Em2.ControlNodes".SemiAutuSplice."step".transition[301],
                          PT := #SeqDelayTime);
   IF #statTonTimer[301].Q THEN
       "Unit1.Em2.ControlNodes".SemiAutuSplice.sequence.status.nextStep := #JOB_3_STEP_03;
   END_IF;
END_REGION

REGION Network 18: Step[303] : Electrode Holder Mover HomePos Check
   RUNG wire#powerrail
      { S7_Templates := "SrcType := DInt" } EQ_Contact(in1 := "Unit1.Em2.ControlNodes".SemiAutuSplice.sequence.status.currentStep, in2 := #JOB_3_STEP_03)
      Contact( "Unit1.Em2.ControlNodes".SemiAutuSplice.sequence.status.seqActive )
      wire#w1
      I_Contact( "Unit1.Em2.ControlNodes".cmElectrodeLeftHolderMoverFwdBwd.monitoring.inWorkPos )
      wire#w2
      Coil( "Unit1.Em2.ControlNodes".SemiAutuSplice."step".action[303] )
   END_RUNG
   RUNG wire#w1
      I_Contact( "Unit1.Em2.ControlNodes".cmElectrodeRightHolderMoverFwdBwd.monitoring.inHomePos )
   END_RUNG wire#w2
   RUNG wire#w1
      Contact( "Unit1.Em2.ControlNodes".cmElectrodeLeftHolderMoverFwdBwd.monitoring.inWorkPos )
      Contact( "Unit1.Em2.ControlNodes".cmElectrodeRightHolderMoverFwdBwd.monitoring.inHomePos )
      Coil( "Unit1.Em2.ControlNodes".SemiAutuSplice."step".transition[303] )
   END_RUNG
   RUNG wire#w1
      Contact( "Unit1.Em2.ControlNodes".SemiAutuSplice."step".transition[303] )
      { S7_Templates := "time_type := Time" } #statTonTimer[303].TON(pt := #SeqDelayTime, et =>)
      Move(in := #JOB_3_STEP_11, out1 => "Unit1.Em2.ControlNodes".SemiAutuSplice.sequence.status.nextStep)
   END_RUNG
   // the same network as SCL:
   #_w1 := ("Unit1.Em2.ControlNodes".SemiAutuSplice.sequence.status.currentStep = #JOB_3_STEP_03) AND "Unit1.Em2.ControlNodes".SemiAutuSplice.sequence.status.seqActive;
   "Unit1.Em2.ControlNodes".SemiAutuSplice."step".action[303] := #_w1 AND (NOT "Unit1.Em2.ControlNodes".cmElectrodeLeftHolderMoverFwdBwd.monitoring.inWorkPos OR NOT "Unit1.Em2.ControlNodes".cmElectrodeRightHolderMoverFwdBwd.monitoring.inHomePos);
   "Unit1.Em2.ControlNodes".SemiAutuSplice."step".transition[303] := #_w1 AND "Unit1.Em2.ControlNodes".cmElectrodeLeftHolderMoverFwdBwd.monitoring.inWorkPos AND "Unit1.Em2.ControlNodes".cmElectrodeRightHolderMoverFwdBwd.monitoring.inHomePos;
   #statTonTimer[303].TON(IN := #_w1 AND "Unit1.Em2.ControlNodes".SemiAutuSplice."step".transition[303],
                          PT := #SeqDelayTime);
   IF #statTonTimer[303].Q THEN
       "Unit1.Em2.ControlNodes".SemiAutuSplice.sequence.status.nextStep := #JOB_3_STEP_11;
   END_IF;
END_REGION

REGION Network 19: Step[311] : Support Unit Shaft Pos Check
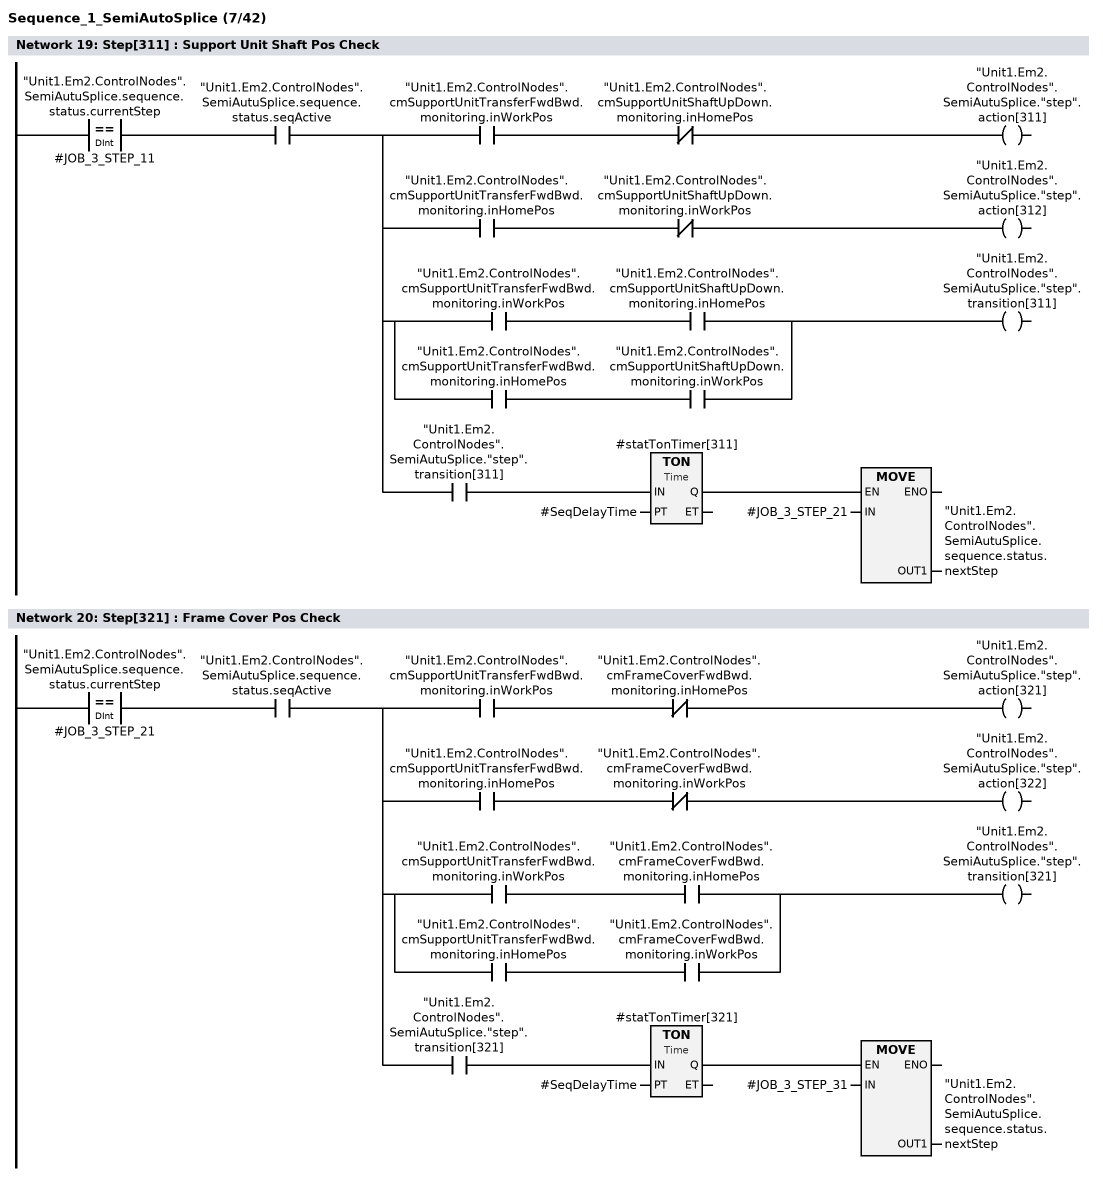
   RUNG wire#powerrail
      { S7_Templates := "SrcType := DInt" } EQ_Contact(in1 := "Unit1.Em2.ControlNodes".SemiAutuSplice.sequence.status.currentStep, in2 := #JOB_3_STEP_11)
      Contact( "Unit1.Em2.ControlNodes".SemiAutuSplice.sequence.status.seqActive )
      wire#w1
      Contact( "Unit1.Em2.ControlNodes".cmSupportUnitTransferFwdBwd.monitoring.inWorkPos )
      I_Contact( "Unit1.Em2.ControlNodes".cmSupportUnitShaftUpDown.monitoring.inHomePos )
      Coil( "Unit1.Em2.ControlNodes".SemiAutuSplice."step".action[311] )
   END_RUNG
   RUNG wire#w1
      Contact( "Unit1.Em2.ControlNodes".cmSupportUnitTransferFwdBwd.monitoring.inHomePos )
      I_Contact( "Unit1.Em2.ControlNodes".cmSupportUnitShaftUpDown.monitoring.inWorkPos )
      Coil( "Unit1.Em2.ControlNodes".SemiAutuSplice."step".action[312] )
   END_RUNG
   RUNG wire#w1
      Contact( "Unit1.Em2.ControlNodes".cmSupportUnitTransferFwdBwd.monitoring.inWorkPos )
      Contact( "Unit1.Em2.ControlNodes".cmSupportUnitShaftUpDown.monitoring.inHomePos )
      wire#w2
      Coil( "Unit1.Em2.ControlNodes".SemiAutuSplice."step".transition[311] )
   END_RUNG
   RUNG wire#w1
      Contact( "Unit1.Em2.ControlNodes".cmSupportUnitTransferFwdBwd.monitoring.inHomePos )
      Contact( "Unit1.Em2.ControlNodes".cmSupportUnitShaftUpDown.monitoring.inWorkPos )
   END_RUNG wire#w2
   RUNG wire#w1
      Contact( "Unit1.Em2.ControlNodes".SemiAutuSplice."step".transition[311] )
      { S7_Templates := "time_type := Time" } #statTonTimer[311].TON(pt := #SeqDelayTime, et =>)
      Move(in := #JOB_3_STEP_21, out1 => "Unit1.Em2.ControlNodes".SemiAutuSplice.sequence.status.nextStep)
   END_RUNG
   // the same network as SCL:
   #_w1 := ("Unit1.Em2.ControlNodes".SemiAutuSplice.sequence.status.currentStep = #JOB_3_STEP_11) AND "Unit1.Em2.ControlNodes".SemiAutuSplice.sequence.status.seqActive;
   "Unit1.Em2.ControlNodes".SemiAutuSplice."step".action[311] := #_w1 AND "Unit1.Em2.ControlNodes".cmSupportUnitTransferFwdBwd.monitoring.inWorkPos AND NOT "Unit1.Em2.ControlNodes".cmSupportUnitShaftUpDown.monitoring.inHomePos;
   "Unit1.Em2.ControlNodes".SemiAutuSplice."step".action[312] := #_w1 AND "Unit1.Em2.ControlNodes".cmSupportUnitTransferFwdBwd.monitoring.inHomePos AND NOT "Unit1.Em2.ControlNodes".cmSupportUnitShaftUpDown.monitoring.inWorkPos;
   "Unit1.Em2.ControlNodes".SemiAutuSplice."step".transition[311] := #_w1 AND (("Unit1.Em2.ControlNodes".cmSupportUnitTransferFwdBwd.monitoring.inWorkPos AND "Unit1.Em2.ControlNodes".cmSupportUnitShaftUpDown.monitoring.inHomePos) OR ("Unit1.Em2.ControlNodes".cmSupportUnitTransferFwdBwd.monitoring.inHomePos AND "Unit1.Em2.ControlNodes".cmSupportUnitShaftUpDown.monitoring.inWorkPos));
   #statTonTimer[311].TON(IN := #_w1 AND "Unit1.Em2.ControlNodes".SemiAutuSplice."step".transition[311],
                          PT := #SeqDelayTime);
   IF #statTonTimer[311].Q THEN
       "Unit1.Em2.ControlNodes".SemiAutuSplice.sequence.status.nextStep := #JOB_3_STEP_21;
   END_IF;
END_REGION

REGION Network 20: Step[321] : Frame Cover Pos Check
   RUNG wire#powerrail
      { S7_Templates := "SrcType := DInt" } EQ_Contact(in1 := "Unit1.Em2.ControlNodes".SemiAutuSplice.sequence.status.currentStep, in2 := #JOB_3_STEP_21)
      Contact( "Unit1.Em2.ControlNodes".SemiAutuSplice.sequence.status.seqActive )
      wire#w1
      Contact( "Unit1.Em2.ControlNodes".cmSupportUnitTransferFwdBwd.monitoring.inWorkPos )
      I_Contact( "Unit1.Em2.ControlNodes".cmFrameCoverFwdBwd.monitoring.inHomePos )
      Coil( "Unit1.Em2.ControlNodes".SemiAutuSplice."step".action[321] )
   END_RUNG
   RUNG wire#w1
      Contact( "Unit1.Em2.ControlNodes".cmSupportUnitTransferFwdBwd.monitoring.inHomePos )
      I_Contact( "Unit1.Em2.ControlNodes".cmFrameCoverFwdBwd.monitoring.inWorkPos )
      Coil( "Unit1.Em2.ControlNodes".SemiAutuSplice."step".action[322] )
   END_RUNG
   RUNG wire#w1
      Contact( "Unit1.Em2.ControlNodes".cmSupportUnitTransferFwdBwd.monitoring.inWorkPos )
      Contact( "Unit1.Em2.ControlNodes".cmFrameCoverFwdBwd.monitoring.inHomePos )
      wire#w2
      Coil( "Unit1.Em2.ControlNodes".SemiAutuSplice."step".transition[321] )
   END_RUNG
   RUNG wire#w1
      Contact( "Unit1.Em2.ControlNodes".cmSupportUnitTransferFwdBwd.monitoring.inHomePos )
      Contact( "Unit1.Em2.ControlNodes".cmFrameCoverFwdBwd.monitoring.inWorkPos )
   END_RUNG wire#w2
   RUNG wire#w1
      Contact( "Unit1.Em2.ControlNodes".SemiAutuSplice."step".transition[321] )
      { S7_Templates := "time_type := Time" } #statTonTimer[321].TON(pt := #SeqDelayTime, et =>)
      Move(in := #JOB_3_STEP_31, out1 => "Unit1.Em2.ControlNodes".SemiAutuSplice.sequence.status.nextStep)
   END_RUNG
   // the same network as SCL:
   #_w1 := ("Unit1.Em2.ControlNodes".SemiAutuSplice.sequence.status.currentStep = #JOB_3_STEP_21) AND "Unit1.Em2.ControlNodes".SemiAutuSplice.sequence.status.seqActive;
   "Unit1.Em2.ControlNodes".SemiAutuSplice."step".action[321] := #_w1 AND "Unit1.Em2.ControlNodes".cmSupportUnitTransferFwdBwd.monitoring.inWorkPos AND NOT "Unit1.Em2.ControlNodes".cmFrameCoverFwdBwd.monitoring.inHomePos;
   "Unit1.Em2.ControlNodes".SemiAutuSplice."step".action[322] := #_w1 AND "Unit1.Em2.ControlNodes".cmSupportUnitTransferFwdBwd.monitoring.inHomePos AND NOT "Unit1.Em2.ControlNodes".cmFrameCoverFwdBwd.monitoring.inWorkPos;
   "Unit1.Em2.ControlNodes".SemiAutuSplice."step".transition[321] := #_w1 AND (("Unit1.Em2.ControlNodes".cmSupportUnitTransferFwdBwd.monitoring.inWorkPos AND "Unit1.Em2.ControlNodes".cmFrameCoverFwdBwd.monitoring.inHomePos) OR ("Unit1.Em2.ControlNodes".cmSupportUnitTransferFwdBwd.monitoring.inHomePos AND "Unit1.Em2.ControlNodes".cmFrameCoverFwdBwd.monitoring.inWorkPos));
   #statTonTimer[321].TON(IN := #_w1 AND "Unit1.Em2.ControlNodes".SemiAutuSplice."step".transition[321],
                          PT := #SeqDelayTime);
   IF #statTonTimer[321].Q THEN
       "Unit1.Em2.ControlNodes".SemiAutuSplice.sequence.status.nextStep := #JOB_3_STEP_31;
   END_IF;
END_REGION

REGION Network 21: Step[331] : Support Unit Transfer HomePos Check
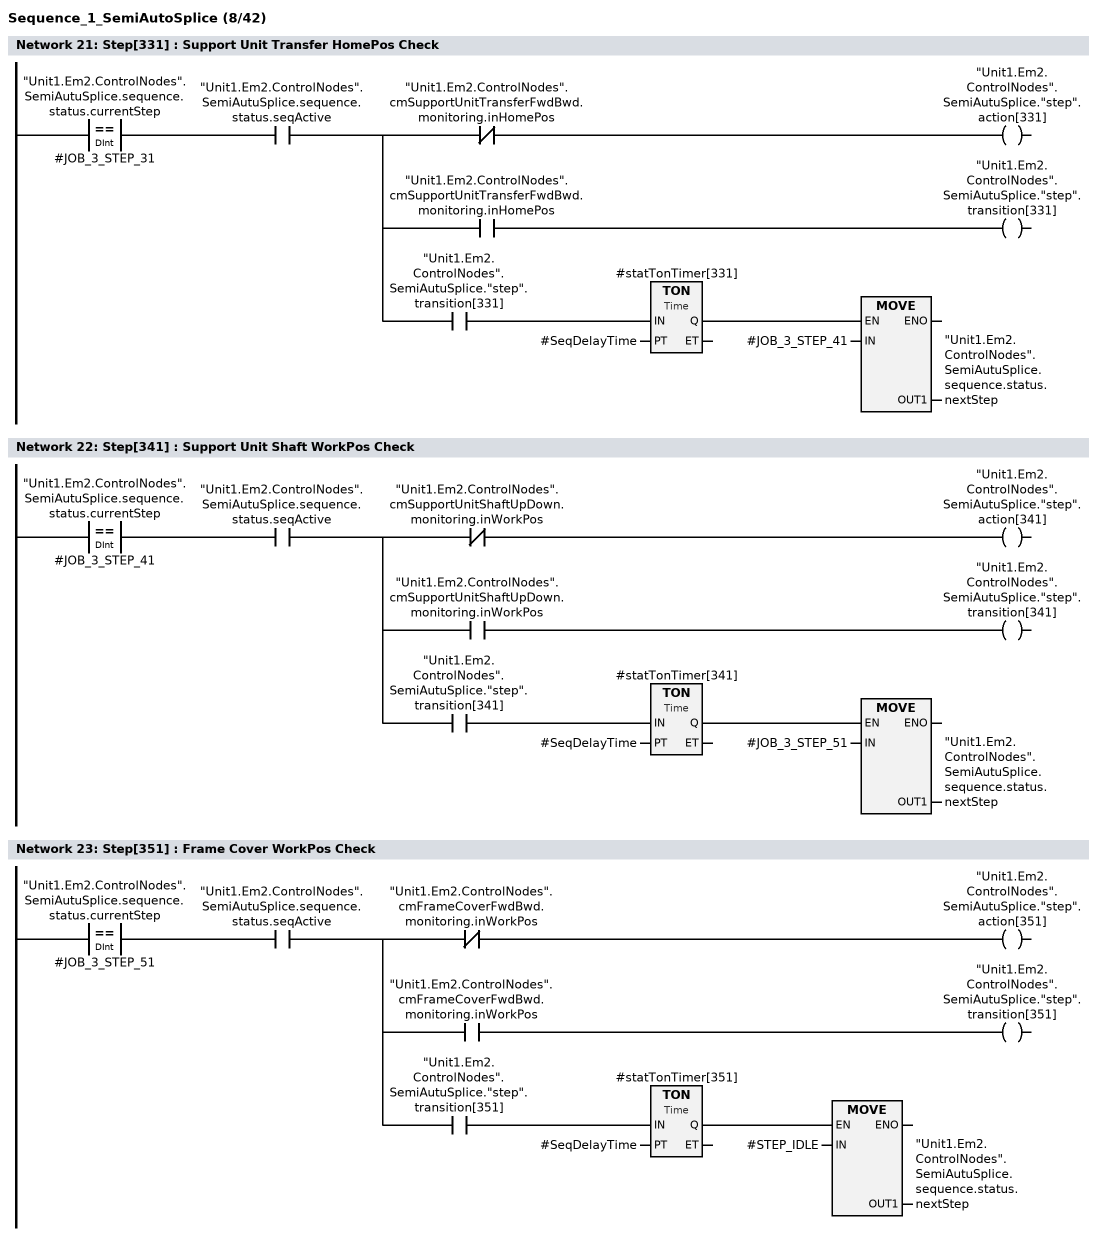
   RUNG wire#powerrail
      { S7_Templates := "SrcType := DInt" } EQ_Contact(in1 := "Unit1.Em2.ControlNodes".SemiAutuSplice.sequence.status.currentStep, in2 := #JOB_3_STEP_31)
      Contact( "Unit1.Em2.ControlNodes".SemiAutuSplice.sequence.status.seqActive )
      wire#w1
      I_Contact( "Unit1.Em2.ControlNodes".cmSupportUnitTransferFwdBwd.monitoring.inHomePos )
      Coil( "Unit1.Em2.ControlNodes".SemiAutuSplice."step".action[331] )
   END_RUNG
   RUNG wire#w1
      Contact( "Unit1.Em2.ControlNodes".cmSupportUnitTransferFwdBwd.monitoring.inHomePos )
      Coil( "Unit1.Em2.ControlNodes".SemiAutuSplice."step".transition[331] )
   END_RUNG
   RUNG wire#w1
      Contact( "Unit1.Em2.ControlNodes".SemiAutuSplice."step".transition[331] )
      { S7_Templates := "time_type := Time" } #statTonTimer[331].TON(pt := #SeqDelayTime, et =>)
      Move(in := #JOB_3_STEP_41, out1 => "Unit1.Em2.ControlNodes".SemiAutuSplice.sequence.status.nextStep)
   END_RUNG
   // the same network as SCL:
   #_w1 := ("Unit1.Em2.ControlNodes".SemiAutuSplice.sequence.status.currentStep = #JOB_3_STEP_31) AND "Unit1.Em2.ControlNodes".SemiAutuSplice.sequence.status.seqActive;
   "Unit1.Em2.ControlNodes".SemiAutuSplice."step".action[331] := #_w1 AND NOT "Unit1.Em2.ControlNodes".cmSupportUnitTransferFwdBwd.monitoring.inHomePos;
   "Unit1.Em2.ControlNodes".SemiAutuSplice."step".transition[331] := #_w1 AND "Unit1.Em2.ControlNodes".cmSupportUnitTransferFwdBwd.monitoring.inHomePos;
   #statTonTimer[331].TON(IN := #_w1 AND "Unit1.Em2.ControlNodes".SemiAutuSplice."step".transition[331],
                          PT := #SeqDelayTime);
   IF #statTonTimer[331].Q THEN
       "Unit1.Em2.ControlNodes".SemiAutuSplice.sequence.status.nextStep := #JOB_3_STEP_41;
   END_IF;
END_REGION

REGION Network 22: Step[341] : Support Unit Shaft WorkPos Check
   RUNG wire#powerrail
      { S7_Templates := "SrcType := DInt" } EQ_Contact(in1 := "Unit1.Em2.ControlNodes".SemiAutuSplice.sequence.status.currentStep, in2 := #JOB_3_STEP_41)
      Contact( "Unit1.Em2.ControlNodes".SemiAutuSplice.sequence.status.seqActive )
      wire#w1
      I_Contact( "Unit1.Em2.ControlNodes".cmSupportUnitShaftUpDown.monitoring.inWorkPos )
      Coil( "Unit1.Em2.ControlNodes".SemiAutuSplice."step".action[341] )
   END_RUNG
   RUNG wire#w1
      Contact( "Unit1.Em2.ControlNodes".cmSupportUnitShaftUpDown.monitoring.inWorkPos )
      Coil( "Unit1.Em2.ControlNodes".SemiAutuSplice."step".transition[341] )
   END_RUNG
   RUNG wire#w1
      Contact( "Unit1.Em2.ControlNodes".SemiAutuSplice."step".transition[341] )
      { S7_Templates := "time_type := Time" } #statTonTimer[341].TON(pt := #SeqDelayTime, et =>)
      Move(in := #JOB_3_STEP_51, out1 => "Unit1.Em2.ControlNodes".SemiAutuSplice.sequence.status.nextStep)
   END_RUNG
   // the same network as SCL:
   #_w1 := ("Unit1.Em2.ControlNodes".SemiAutuSplice.sequence.status.currentStep = #JOB_3_STEP_41) AND "Unit1.Em2.ControlNodes".SemiAutuSplice.sequence.status.seqActive;
   "Unit1.Em2.ControlNodes".SemiAutuSplice."step".action[341] := #_w1 AND NOT "Unit1.Em2.ControlNodes".cmSupportUnitShaftUpDown.monitoring.inWorkPos;
   "Unit1.Em2.ControlNodes".SemiAutuSplice."step".transition[341] := #_w1 AND "Unit1.Em2.ControlNodes".cmSupportUnitShaftUpDown.monitoring.inWorkPos;
   #statTonTimer[341].TON(IN := #_w1 AND "Unit1.Em2.ControlNodes".SemiAutuSplice."step".transition[341],
                          PT := #SeqDelayTime);
   IF #statTonTimer[341].Q THEN
       "Unit1.Em2.ControlNodes".SemiAutuSplice.sequence.status.nextStep := #JOB_3_STEP_51;
   END_IF;
END_REGION

REGION Network 23: Step[351] : Frame Cover WorkPos Check
   RUNG wire#powerrail
      { S7_Templates := "SrcType := DInt" } EQ_Contact(in1 := "Unit1.Em2.ControlNodes".SemiAutuSplice.sequence.status.currentStep, in2 := #JOB_3_STEP_51)
      Contact( "Unit1.Em2.ControlNodes".SemiAutuSplice.sequence.status.seqActive )
      wire#w1
      I_Contact( "Unit1.Em2.ControlNodes".cmFrameCoverFwdBwd.monitoring.inWorkPos )
      Coil( "Unit1.Em2.ControlNodes".SemiAutuSplice."step".action[351] )
   END_RUNG
   RUNG wire#w1
      Contact( "Unit1.Em2.ControlNodes".cmFrameCoverFwdBwd.monitoring.inWorkPos )
      Coil( "Unit1.Em2.ControlNodes".SemiAutuSplice."step".transition[351] )
   END_RUNG
   RUNG wire#w1
      Contact( "Unit1.Em2.ControlNodes".SemiAutuSplice."step".transition[351] )
      { S7_Templates := "time_type := Time" } #statTonTimer[351].TON(pt := #SeqDelayTime, et =>)
      Move(in := #STEP_IDLE, out1 => "Unit1.Em2.ControlNodes".SemiAutuSplice.sequence.status.nextStep)
   END_RUNG
   // the same network as SCL:
   #_w1 := ("Unit1.Em2.ControlNodes".SemiAutuSplice.sequence.status.currentStep = #JOB_3_STEP_51) AND "Unit1.Em2.ControlNodes".SemiAutuSplice.sequence.status.seqActive;
   "Unit1.Em2.ControlNodes".SemiAutuSplice."step".action[351] := #_w1 AND NOT "Unit1.Em2.ControlNodes".cmFrameCoverFwdBwd.monitoring.inWorkPos;
   "Unit1.Em2.ControlNodes".SemiAutuSplice."step".transition[351] := #_w1 AND "Unit1.Em2.ControlNodes".cmFrameCoverFwdBwd.monitoring.inWorkPos;
   #statTonTimer[351].TON(IN := #_w1 AND "Unit1.Em2.ControlNodes".SemiAutuSplice."step".transition[351],
                          PT := #SeqDelayTime);
   IF #statTonTimer[351].Q THEN
       "Unit1.Em2.ControlNodes".SemiAutuSplice.sequence.status.nextStep := #STEP_IDLE;
   END_IF;
END_REGION

REGION Network 24: ******************** JOB[4] RIGHT SPLICING MODULE MOVER INITIALIZED ********************
END_REGION

REGION Network 25: Step[401] : Splicing Left & Right Module Mover HomePos Check
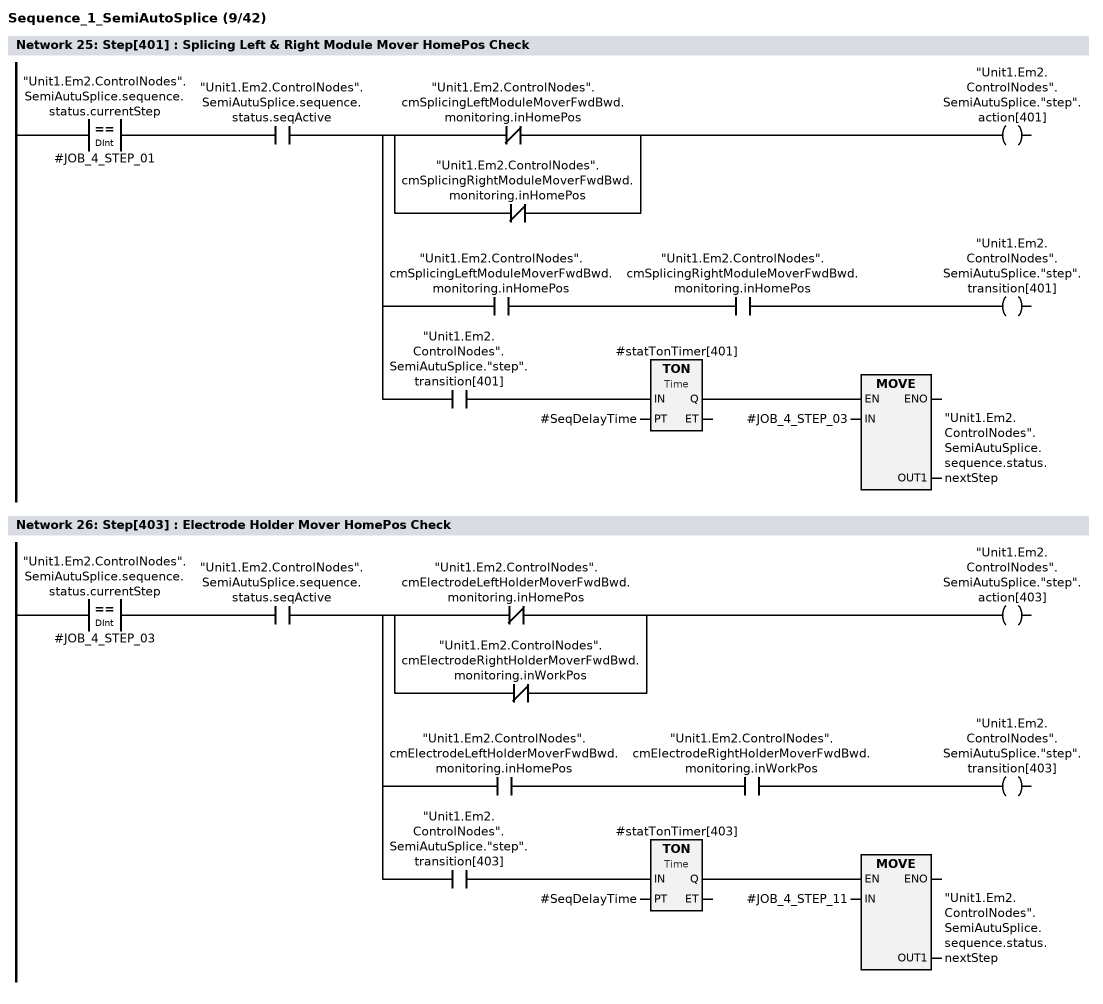
   RUNG wire#powerrail
      { S7_Templates := "SrcType := DInt" } EQ_Contact(in1 := "Unit1.Em2.ControlNodes".SemiAutuSplice.sequence.status.currentStep, in2 := #JOB_4_STEP_01)
      Contact( "Unit1.Em2.ControlNodes".SemiAutuSplice.sequence.status.seqActive )
      wire#w1
      I_Contact( "Unit1.Em2.ControlNodes".cmSplicingLeftModuleMoverFwdBwd.monitoring.inHomePos )
      wire#w2
      Coil( "Unit1.Em2.ControlNodes".SemiAutuSplice."step".action[401] )
   END_RUNG
   RUNG wire#w1
      I_Contact( "Unit1.Em2.ControlNodes".cmSplicingRightModuleMoverFwdBwd.monitoring.inHomePos )
   END_RUNG wire#w2
   RUNG wire#w1
      Contact( "Unit1.Em2.ControlNodes".cmSplicingLeftModuleMoverFwdBwd.monitoring.inHomePos )
      Contact( "Unit1.Em2.ControlNodes".cmSplicingRightModuleMoverFwdBwd.monitoring.inHomePos )
      Coil( "Unit1.Em2.ControlNodes".SemiAutuSplice."step".transition[401] )
   END_RUNG
   RUNG wire#w1
      Contact( "Unit1.Em2.ControlNodes".SemiAutuSplice."step".transition[401] )
      { S7_Templates := "time_type := Time" } #statTonTimer[401].TON(pt := #SeqDelayTime, et =>)
      Move(in := #JOB_4_STEP_03, out1 => "Unit1.Em2.ControlNodes".SemiAutuSplice.sequence.status.nextStep)
   END_RUNG
   // the same network as SCL:
   #_w1 := ("Unit1.Em2.ControlNodes".SemiAutuSplice.sequence.status.currentStep = #JOB_4_STEP_01) AND "Unit1.Em2.ControlNodes".SemiAutuSplice.sequence.status.seqActive;
   "Unit1.Em2.ControlNodes".SemiAutuSplice."step".action[401] := #_w1 AND (NOT "Unit1.Em2.ControlNodes".cmSplicingLeftModuleMoverFwdBwd.monitoring.inHomePos OR NOT "Unit1.Em2.ControlNodes".cmSplicingRightModuleMoverFwdBwd.monitoring.inHomePos);
   "Unit1.Em2.ControlNodes".SemiAutuSplice."step".transition[401] := #_w1 AND "Unit1.Em2.ControlNodes".cmSplicingLeftModuleMoverFwdBwd.monitoring.inHomePos AND "Unit1.Em2.ControlNodes".cmSplicingRightModuleMoverFwdBwd.monitoring.inHomePos;
   #statTonTimer[401].TON(IN := #_w1 AND "Unit1.Em2.ControlNodes".SemiAutuSplice."step".transition[401],
                          PT := #SeqDelayTime);
   IF #statTonTimer[401].Q THEN
       "Unit1.Em2.ControlNodes".SemiAutuSplice.sequence.status.nextStep := #JOB_4_STEP_03;
   END_IF;
END_REGION

REGION Network 26: Step[403] : Electrode Holder Mover HomePos Check
   RUNG wire#powerrail
      { S7_Templates := "SrcType := DInt" } EQ_Contact(in1 := "Unit1.Em2.ControlNodes".SemiAutuSplice.sequence.status.currentStep, in2 := #JOB_4_STEP_03)
      Contact( "Unit1.Em2.ControlNodes".SemiAutuSplice.sequence.status.seqActive )
      wire#w1
      I_Contact( "Unit1.Em2.ControlNodes".cmElectrodeLeftHolderMoverFwdBwd.monitoring.inHomePos )
      wire#w2
      Coil( "Unit1.Em2.ControlNodes".SemiAutuSplice."step".action[403] )
   END_RUNG
   RUNG wire#w1
      I_Contact( "Unit1.Em2.ControlNodes".cmElectrodeRightHolderMoverFwdBwd.monitoring.inWorkPos )
   END_RUNG wire#w2
   RUNG wire#w1
      Contact( "Unit1.Em2.ControlNodes".cmElectrodeLeftHolderMoverFwdBwd.monitoring.inHomePos )
      Contact( "Unit1.Em2.ControlNodes".cmElectrodeRightHolderMoverFwdBwd.monitoring.inWorkPos )
      Coil( "Unit1.Em2.ControlNodes".SemiAutuSplice."step".transition[403] )
   END_RUNG
   RUNG wire#w1
      Contact( "Unit1.Em2.ControlNodes".SemiAutuSplice."step".transition[403] )
      { S7_Templates := "time_type := Time" } #statTonTimer[403].TON(pt := #SeqDelayTime, et =>)
      Move(in := #JOB_4_STEP_11, out1 => "Unit1.Em2.ControlNodes".SemiAutuSplice.sequence.status.nextStep)
   END_RUNG
   // the same network as SCL:
   #_w1 := ("Unit1.Em2.ControlNodes".SemiAutuSplice.sequence.status.currentStep = #JOB_4_STEP_03) AND "Unit1.Em2.ControlNodes".SemiAutuSplice.sequence.status.seqActive;
   "Unit1.Em2.ControlNodes".SemiAutuSplice."step".action[403] := #_w1 AND (NOT "Unit1.Em2.ControlNodes".cmElectrodeLeftHolderMoverFwdBwd.monitoring.inHomePos OR NOT "Unit1.Em2.ControlNodes".cmElectrodeRightHolderMoverFwdBwd.monitoring.inWorkPos);
   "Unit1.Em2.ControlNodes".SemiAutuSplice."step".transition[403] := #_w1 AND "Unit1.Em2.ControlNodes".cmElectrodeLeftHolderMoverFwdBwd.monitoring.inHomePos AND "Unit1.Em2.ControlNodes".cmElectrodeRightHolderMoverFwdBwd.monitoring.inWorkPos;
   #statTonTimer[403].TON(IN := #_w1 AND "Unit1.Em2.ControlNodes".SemiAutuSplice."step".transition[403],
                          PT := #SeqDelayTime);
   IF #statTonTimer[403].Q THEN
       "Unit1.Em2.ControlNodes".SemiAutuSplice.sequence.status.nextStep := #JOB_4_STEP_11;
   END_IF;
END_REGION

REGION Network 27: Step[411] : Support Unit Shaft Pos Check
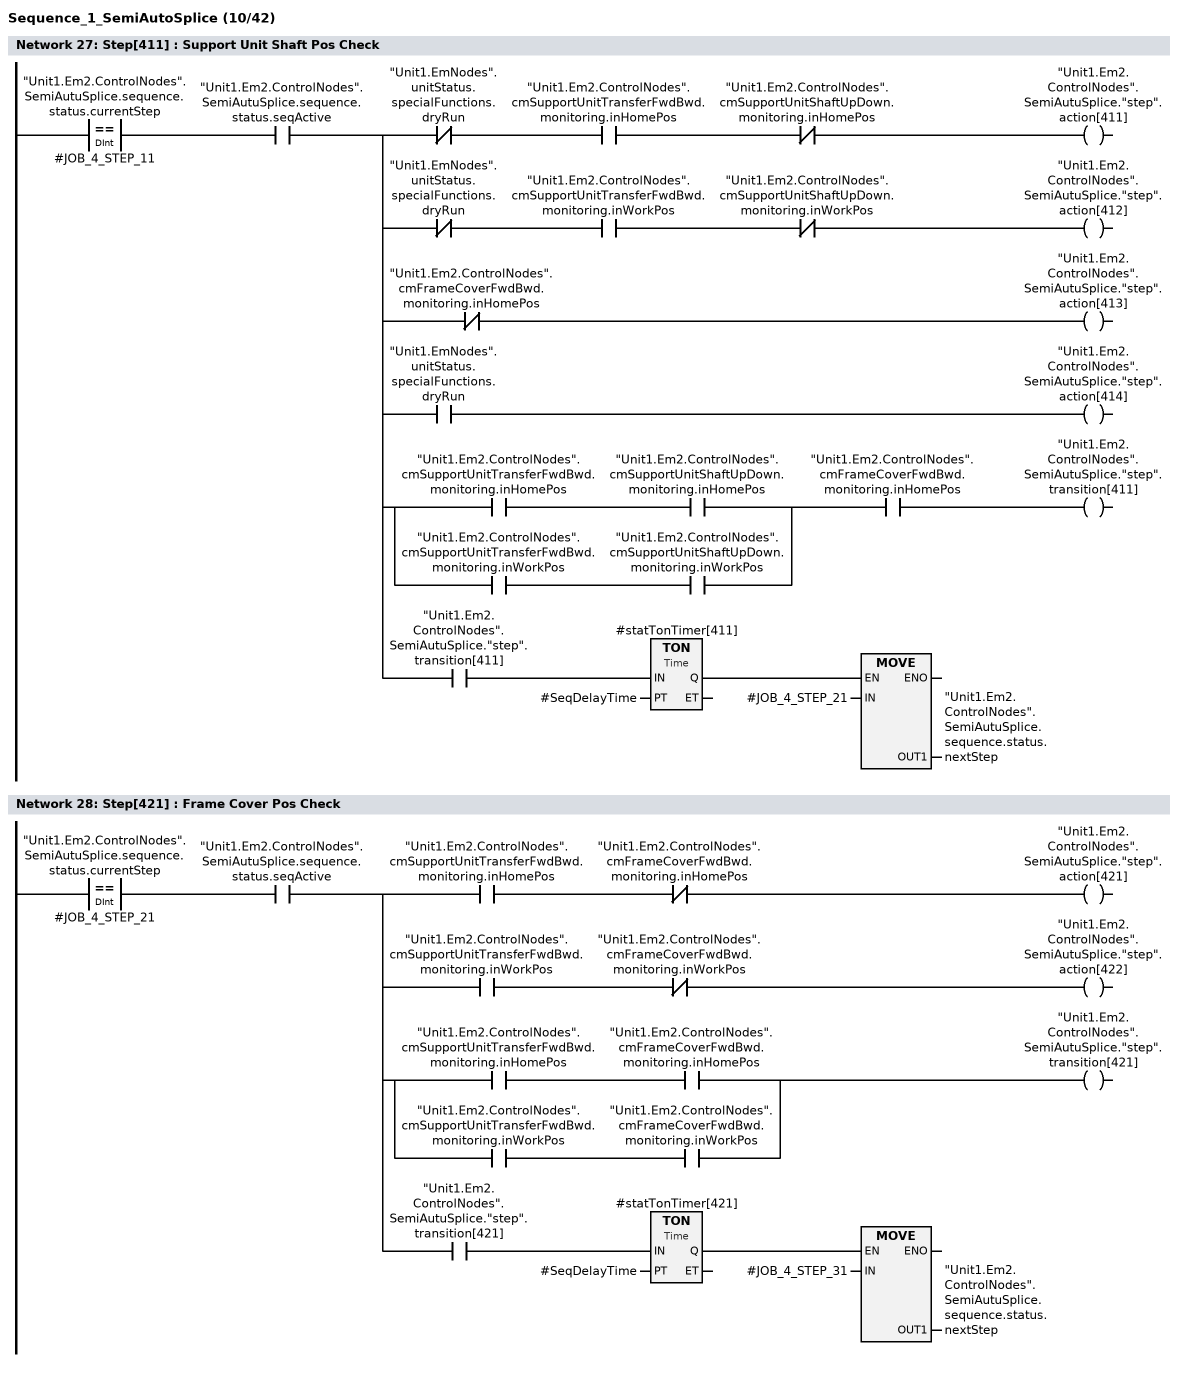
   RUNG wire#powerrail
      { S7_Templates := "SrcType := DInt" } EQ_Contact(in1 := "Unit1.Em2.ControlNodes".SemiAutuSplice.sequence.status.currentStep, in2 := #JOB_4_STEP_11)
      Contact( "Unit1.Em2.ControlNodes".SemiAutuSplice.sequence.status.seqActive )
      wire#w1
      I_Contact( "Unit1.EmNodes".unitStatus.specialFunctions.dryRun )
      Contact( "Unit1.Em2.ControlNodes".cmSupportUnitTransferFwdBwd.monitoring.inHomePos )
      I_Contact( "Unit1.Em2.ControlNodes".cmSupportUnitShaftUpDown.monitoring.inHomePos )
      Coil( "Unit1.Em2.ControlNodes".SemiAutuSplice."step".action[411] )
   END_RUNG
   RUNG wire#w1
      I_Contact( "Unit1.EmNodes".unitStatus.specialFunctions.dryRun )
      Contact( "Unit1.Em2.ControlNodes".cmSupportUnitTransferFwdBwd.monitoring.inWorkPos )
      I_Contact( "Unit1.Em2.ControlNodes".cmSupportUnitShaftUpDown.monitoring.inWorkPos )
      Coil( "Unit1.Em2.ControlNodes".SemiAutuSplice."step".action[412] )
   END_RUNG
   RUNG wire#w1
      I_Contact( "Unit1.Em2.ControlNodes".cmFrameCoverFwdBwd.monitoring.inHomePos )
      Coil( "Unit1.Em2.ControlNodes".SemiAutuSplice."step".action[413] )
   END_RUNG
   RUNG wire#w1
      Contact( "Unit1.EmNodes".unitStatus.specialFunctions.dryRun )
      Coil( "Unit1.Em2.ControlNodes".SemiAutuSplice."step".action[414] )
   END_RUNG
   RUNG wire#w1
      Contact( "Unit1.Em2.ControlNodes".cmSupportUnitTransferFwdBwd.monitoring.inHomePos )
      Contact( "Unit1.Em2.ControlNodes".cmSupportUnitShaftUpDown.monitoring.inHomePos )
      wire#w2
      Contact( "Unit1.Em2.ControlNodes".cmFrameCoverFwdBwd.monitoring.inHomePos )
      Coil( "Unit1.Em2.ControlNodes".SemiAutuSplice."step".transition[411] )
   END_RUNG
   RUNG wire#w1
      Contact( "Unit1.Em2.ControlNodes".cmSupportUnitTransferFwdBwd.monitoring.inWorkPos )
      Contact( "Unit1.Em2.ControlNodes".cmSupportUnitShaftUpDown.monitoring.inWorkPos )
   END_RUNG wire#w2
   RUNG wire#w1
      Contact( "Unit1.Em2.ControlNodes".SemiAutuSplice."step".transition[411] )
      { S7_Templates := "time_type := Time" } #statTonTimer[411].TON(pt := #SeqDelayTime, et =>)
      Move(in := #JOB_4_STEP_21, out1 => "Unit1.Em2.ControlNodes".SemiAutuSplice.sequence.status.nextStep)
   END_RUNG
   // the same network as SCL:
   #_w1 := ("Unit1.Em2.ControlNodes".SemiAutuSplice.sequence.status.currentStep = #JOB_4_STEP_11) AND "Unit1.Em2.ControlNodes".SemiAutuSplice.sequence.status.seqActive;
   "Unit1.Em2.ControlNodes".SemiAutuSplice."step".action[411] := #_w1 AND NOT "Unit1.EmNodes".unitStatus.specialFunctions.dryRun AND "Unit1.Em2.ControlNodes".cmSupportUnitTransferFwdBwd.monitoring.inHomePos AND NOT "Unit1.Em2.ControlNodes".cmSupportUnitShaftUpDown.monitoring.inHomePos;
   "Unit1.Em2.ControlNodes".SemiAutuSplice."step".action[412] := #_w1 AND NOT "Unit1.EmNodes".unitStatus.specialFunctions.dryRun AND "Unit1.Em2.ControlNodes".cmSupportUnitTransferFwdBwd.monitoring.inWorkPos AND NOT "Unit1.Em2.ControlNodes".cmSupportUnitShaftUpDown.monitoring.inWorkPos;
   "Unit1.Em2.ControlNodes".SemiAutuSplice."step".action[413] := #_w1 AND NOT "Unit1.Em2.ControlNodes".cmFrameCoverFwdBwd.monitoring.inHomePos;
   "Unit1.Em2.ControlNodes".SemiAutuSplice."step".action[414] := #_w1 AND "Unit1.EmNodes".unitStatus.specialFunctions.dryRun;
   "Unit1.Em2.ControlNodes".SemiAutuSplice."step".transition[411] := #_w1 AND (("Unit1.Em2.ControlNodes".cmSupportUnitTransferFwdBwd.monitoring.inHomePos AND "Unit1.Em2.ControlNodes".cmSupportUnitShaftUpDown.monitoring.inHomePos) OR ("Unit1.Em2.ControlNodes".cmSupportUnitTransferFwdBwd.monitoring.inWorkPos AND "Unit1.Em2.ControlNodes".cmSupportUnitShaftUpDown.monitoring.inWorkPos)) AND "Unit1.Em2.ControlNodes".cmFrameCoverFwdBwd.monitoring.inHomePos;
   #statTonTimer[411].TON(IN := #_w1 AND "Unit1.Em2.ControlNodes".SemiAutuSplice."step".transition[411],
                          PT := #SeqDelayTime);
   IF #statTonTimer[411].Q THEN
       "Unit1.Em2.ControlNodes".SemiAutuSplice.sequence.status.nextStep := #JOB_4_STEP_21;
   END_IF;
END_REGION

REGION Network 28: Step[421] : Frame Cover Pos Check
   RUNG wire#powerrail
      { S7_Templates := "SrcType := DInt" } EQ_Contact(in1 := "Unit1.Em2.ControlNodes".SemiAutuSplice.sequence.status.currentStep, in2 := #JOB_4_STEP_21)
      Contact( "Unit1.Em2.ControlNodes".SemiAutuSplice.sequence.status.seqActive )
      wire#w1
      Contact( "Unit1.Em2.ControlNodes".cmSupportUnitTransferFwdBwd.monitoring.inHomePos )
      I_Contact( "Unit1.Em2.ControlNodes".cmFrameCoverFwdBwd.monitoring.inHomePos )
      Coil( "Unit1.Em2.ControlNodes".SemiAutuSplice."step".action[421] )
   END_RUNG
   RUNG wire#w1
      Contact( "Unit1.Em2.ControlNodes".cmSupportUnitTransferFwdBwd.monitoring.inWorkPos )
      I_Contact( "Unit1.Em2.ControlNodes".cmFrameCoverFwdBwd.monitoring.inWorkPos )
      Coil( "Unit1.Em2.ControlNodes".SemiAutuSplice."step".action[422] )
   END_RUNG
   RUNG wire#w1
      Contact( "Unit1.Em2.ControlNodes".cmSupportUnitTransferFwdBwd.monitoring.inHomePos )
      Contact( "Unit1.Em2.ControlNodes".cmFrameCoverFwdBwd.monitoring.inHomePos )
      wire#w2
      Coil( "Unit1.Em2.ControlNodes".SemiAutuSplice."step".transition[421] )
   END_RUNG
   RUNG wire#w1
      Contact( "Unit1.Em2.ControlNodes".cmSupportUnitTransferFwdBwd.monitoring.inWorkPos )
      Contact( "Unit1.Em2.ControlNodes".cmFrameCoverFwdBwd.monitoring.inWorkPos )
   END_RUNG wire#w2
   RUNG wire#w1
      Contact( "Unit1.Em2.ControlNodes".SemiAutuSplice."step".transition[421] )
      { S7_Templates := "time_type := Time" } #statTonTimer[421].TON(pt := #SeqDelayTime, et =>)
      Move(in := #JOB_4_STEP_31, out1 => "Unit1.Em2.ControlNodes".SemiAutuSplice.sequence.status.nextStep)
   END_RUNG
   // the same network as SCL:
   #_w1 := ("Unit1.Em2.ControlNodes".SemiAutuSplice.sequence.status.currentStep = #JOB_4_STEP_21) AND "Unit1.Em2.ControlNodes".SemiAutuSplice.sequence.status.seqActive;
   "Unit1.Em2.ControlNodes".SemiAutuSplice."step".action[421] := #_w1 AND "Unit1.Em2.ControlNodes".cmSupportUnitTransferFwdBwd.monitoring.inHomePos AND NOT "Unit1.Em2.ControlNodes".cmFrameCoverFwdBwd.monitoring.inHomePos;
   "Unit1.Em2.ControlNodes".SemiAutuSplice."step".action[422] := #_w1 AND "Unit1.Em2.ControlNodes".cmSupportUnitTransferFwdBwd.monitoring.inWorkPos AND NOT "Unit1.Em2.ControlNodes".cmFrameCoverFwdBwd.monitoring.inWorkPos;
   "Unit1.Em2.ControlNodes".SemiAutuSplice."step".transition[421] := #_w1 AND (("Unit1.Em2.ControlNodes".cmSupportUnitTransferFwdBwd.monitoring.inHomePos AND "Unit1.Em2.ControlNodes".cmFrameCoverFwdBwd.monitoring.inHomePos) OR ("Unit1.Em2.ControlNodes".cmSupportUnitTransferFwdBwd.monitoring.inWorkPos AND "Unit1.Em2.ControlNodes".cmFrameCoverFwdBwd.monitoring.inWorkPos));
   #statTonTimer[421].TON(IN := #_w1 AND "Unit1.Em2.ControlNodes".SemiAutuSplice."step".transition[421],
                          PT := #SeqDelayTime);
   IF #statTonTimer[421].Q THEN
       "Unit1.Em2.ControlNodes".SemiAutuSplice.sequence.status.nextStep := #JOB_4_STEP_31;
   END_IF;
END_REGION

REGION Network 29: Step[431] : Support Unit Transfer WorkPos Check
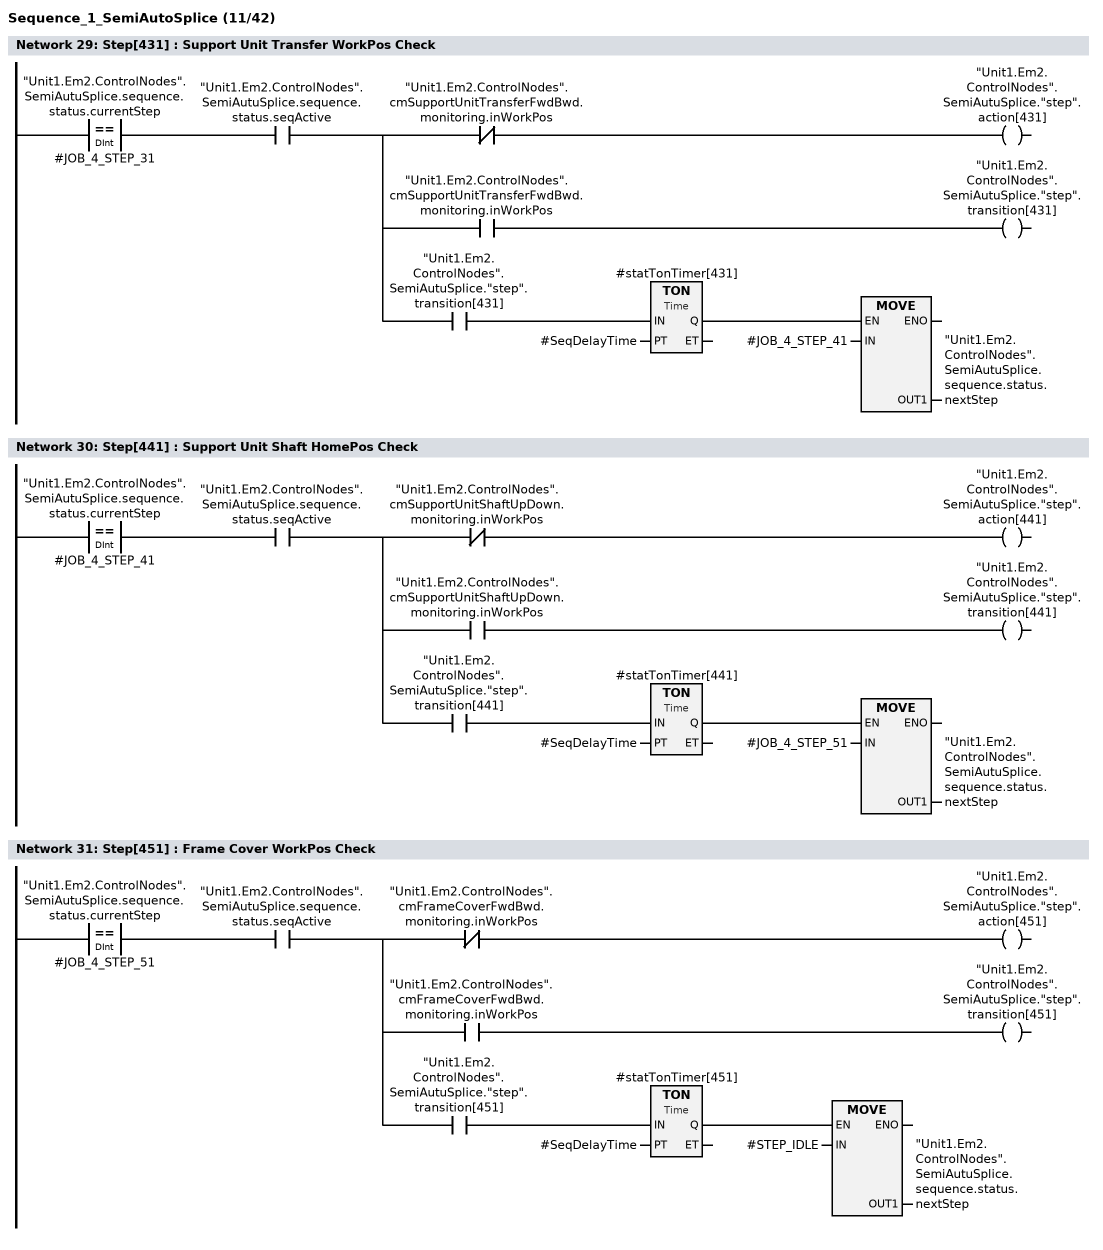
   RUNG wire#powerrail
      { S7_Templates := "SrcType := DInt" } EQ_Contact(in1 := "Unit1.Em2.ControlNodes".SemiAutuSplice.sequence.status.currentStep, in2 := #JOB_4_STEP_31)
      Contact( "Unit1.Em2.ControlNodes".SemiAutuSplice.sequence.status.seqActive )
      wire#w1
      I_Contact( "Unit1.Em2.ControlNodes".cmSupportUnitTransferFwdBwd.monitoring.inWorkPos )
      Coil( "Unit1.Em2.ControlNodes".SemiAutuSplice."step".action[431] )
   END_RUNG
   RUNG wire#w1
      Contact( "Unit1.Em2.ControlNodes".cmSupportUnitTransferFwdBwd.monitoring.inWorkPos )
      Coil( "Unit1.Em2.ControlNodes".SemiAutuSplice."step".transition[431] )
   END_RUNG
   RUNG wire#w1
      Contact( "Unit1.Em2.ControlNodes".SemiAutuSplice."step".transition[431] )
      { S7_Templates := "time_type := Time" } #statTonTimer[431].TON(pt := #SeqDelayTime, et =>)
      Move(in := #JOB_4_STEP_41, out1 => "Unit1.Em2.ControlNodes".SemiAutuSplice.sequence.status.nextStep)
   END_RUNG
   // the same network as SCL:
   #_w1 := ("Unit1.Em2.ControlNodes".SemiAutuSplice.sequence.status.currentStep = #JOB_4_STEP_31) AND "Unit1.Em2.ControlNodes".SemiAutuSplice.sequence.status.seqActive;
   "Unit1.Em2.ControlNodes".SemiAutuSplice."step".action[431] := #_w1 AND NOT "Unit1.Em2.ControlNodes".cmSupportUnitTransferFwdBwd.monitoring.inWorkPos;
   "Unit1.Em2.ControlNodes".SemiAutuSplice."step".transition[431] := #_w1 AND "Unit1.Em2.ControlNodes".cmSupportUnitTransferFwdBwd.monitoring.inWorkPos;
   #statTonTimer[431].TON(IN := #_w1 AND "Unit1.Em2.ControlNodes".SemiAutuSplice."step".transition[431],
                          PT := #SeqDelayTime);
   IF #statTonTimer[431].Q THEN
       "Unit1.Em2.ControlNodes".SemiAutuSplice.sequence.status.nextStep := #JOB_4_STEP_41;
   END_IF;
END_REGION

REGION Network 30: Step[441] : Support Unit Shaft HomePos Check
   RUNG wire#powerrail
      { S7_Templates := "SrcType := DInt" } EQ_Contact(in1 := "Unit1.Em2.ControlNodes".SemiAutuSplice.sequence.status.currentStep, in2 := #JOB_4_STEP_41)
      Contact( "Unit1.Em2.ControlNodes".SemiAutuSplice.sequence.status.seqActive )
      wire#w1
      I_Contact( "Unit1.Em2.ControlNodes".cmSupportUnitShaftUpDown.monitoring.inWorkPos )
      Coil( "Unit1.Em2.ControlNodes".SemiAutuSplice."step".action[441] )
   END_RUNG
   RUNG wire#w1
      Contact( "Unit1.Em2.ControlNodes".cmSupportUnitShaftUpDown.monitoring.inWorkPos )
      Coil( "Unit1.Em2.ControlNodes".SemiAutuSplice."step".transition[441] )
   END_RUNG
   RUNG wire#w1
      Contact( "Unit1.Em2.ControlNodes".SemiAutuSplice."step".transition[441] )
      { S7_Templates := "time_type := Time" } #statTonTimer[441].TON(pt := #SeqDelayTime, et =>)
      Move(in := #JOB_4_STEP_51, out1 => "Unit1.Em2.ControlNodes".SemiAutuSplice.sequence.status.nextStep)
   END_RUNG
   // the same network as SCL:
   #_w1 := ("Unit1.Em2.ControlNodes".SemiAutuSplice.sequence.status.currentStep = #JOB_4_STEP_41) AND "Unit1.Em2.ControlNodes".SemiAutuSplice.sequence.status.seqActive;
   "Unit1.Em2.ControlNodes".SemiAutuSplice."step".action[441] := #_w1 AND NOT "Unit1.Em2.ControlNodes".cmSupportUnitShaftUpDown.monitoring.inWorkPos;
   "Unit1.Em2.ControlNodes".SemiAutuSplice."step".transition[441] := #_w1 AND "Unit1.Em2.ControlNodes".cmSupportUnitShaftUpDown.monitoring.inWorkPos;
   #statTonTimer[441].TON(IN := #_w1 AND "Unit1.Em2.ControlNodes".SemiAutuSplice."step".transition[441],
                          PT := #SeqDelayTime);
   IF #statTonTimer[441].Q THEN
       "Unit1.Em2.ControlNodes".SemiAutuSplice.sequence.status.nextStep := #JOB_4_STEP_51;
   END_IF;
END_REGION

REGION Network 31: Step[451] : Frame Cover WorkPos Check
   RUNG wire#powerrail
      { S7_Templates := "SrcType := DInt" } EQ_Contact(in1 := "Unit1.Em2.ControlNodes".SemiAutuSplice.sequence.status.currentStep, in2 := #JOB_4_STEP_51)
      Contact( "Unit1.Em2.ControlNodes".SemiAutuSplice.sequence.status.seqActive )
      wire#w1
      I_Contact( "Unit1.Em2.ControlNodes".cmFrameCoverFwdBwd.monitoring.inWorkPos )
      Coil( "Unit1.Em2.ControlNodes".SemiAutuSplice."step".action[451] )
   END_RUNG
   RUNG wire#w1
      Contact( "Unit1.Em2.ControlNodes".cmFrameCoverFwdBwd.monitoring.inWorkPos )
      Coil( "Unit1.Em2.ControlNodes".SemiAutuSplice."step".transition[451] )
   END_RUNG
   RUNG wire#w1
      Contact( "Unit1.Em2.ControlNodes".SemiAutuSplice."step".transition[451] )
      { S7_Templates := "time_type := Time" } #statTonTimer[451].TON(pt := #SeqDelayTime, et =>)
      Move(in := #STEP_IDLE, out1 => "Unit1.Em2.ControlNodes".SemiAutuSplice.sequence.status.nextStep)
   END_RUNG
   // the same network as SCL:
   #_w1 := ("Unit1.Em2.ControlNodes".SemiAutuSplice.sequence.status.currentStep = #JOB_4_STEP_51) AND "Unit1.Em2.ControlNodes".SemiAutuSplice.sequence.status.seqActive;
   "Unit1.Em2.ControlNodes".SemiAutuSplice."step".action[451] := #_w1 AND NOT "Unit1.Em2.ControlNodes".cmFrameCoverFwdBwd.monitoring.inWorkPos;
   "Unit1.Em2.ControlNodes".SemiAutuSplice."step".transition[451] := #_w1 AND "Unit1.Em2.ControlNodes".cmFrameCoverFwdBwd.monitoring.inWorkPos;
   #statTonTimer[451].TON(IN := #_w1 AND "Unit1.Em2.ControlNodes".SemiAutuSplice."step".transition[451],
                          PT := #SeqDelayTime);
   IF #statTonTimer[451].Q THEN
       "Unit1.Em2.ControlNodes".SemiAutuSplice.sequence.status.nextStep := #STEP_IDLE;
   END_IF;
END_REGION

REGION Network 32: ******************** JOB[5] SPLICING MODULE MOVER AUTO ********************
END_REGION

REGION Network 33: Step[501] : Splicing Module Mover WorkPos Command
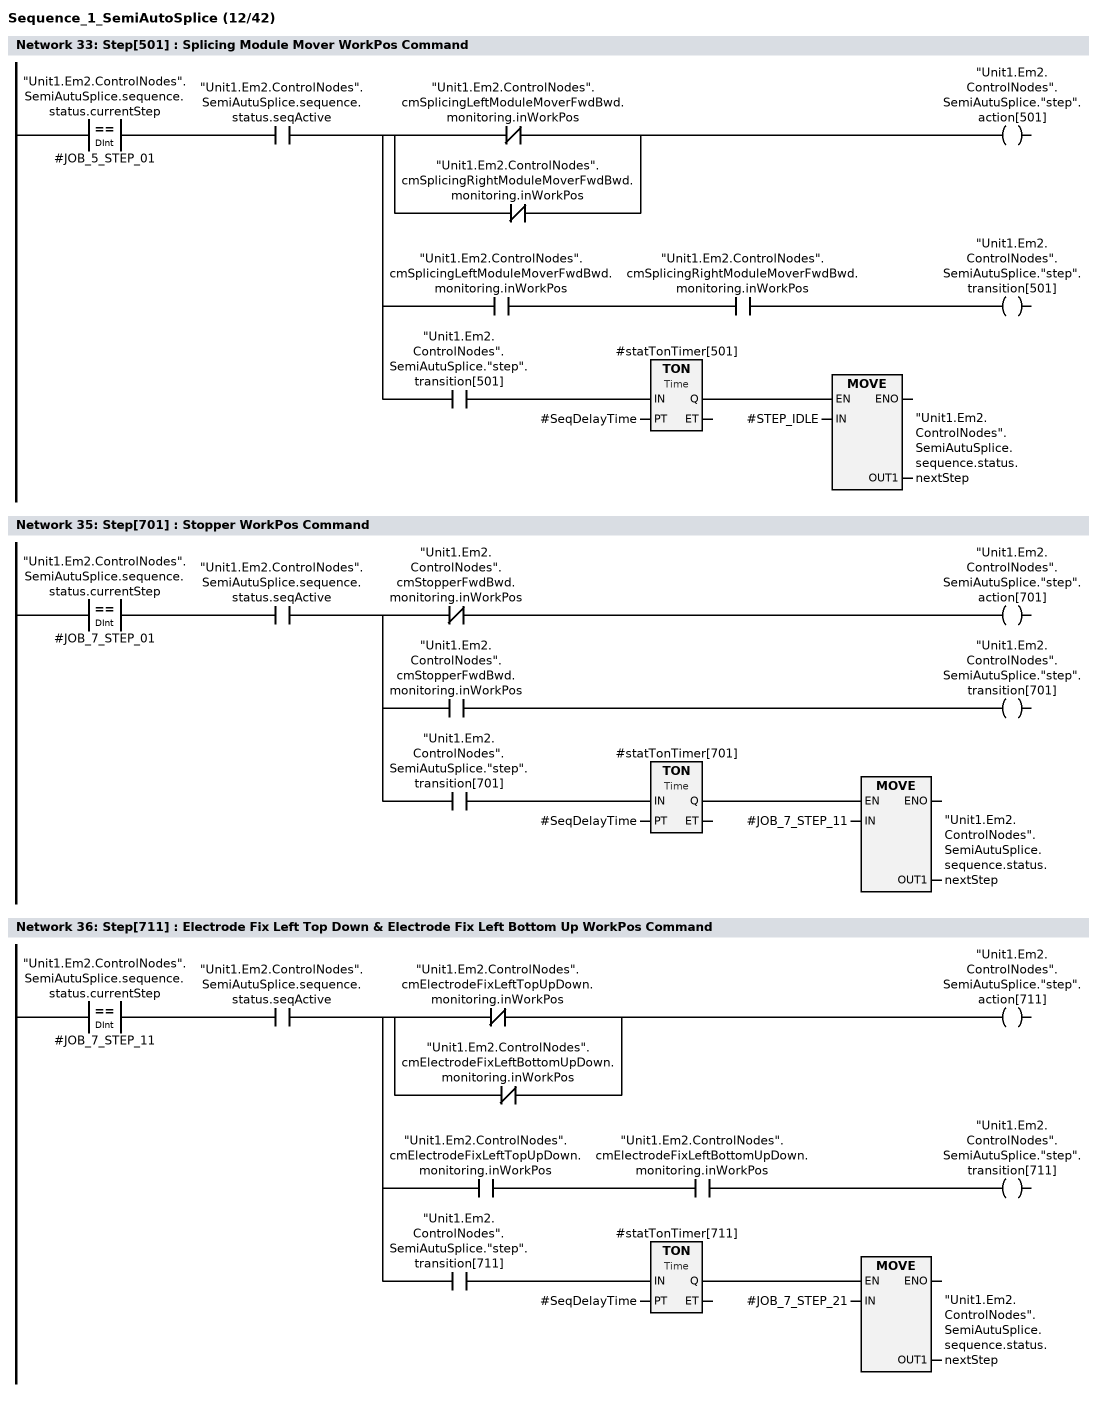
   RUNG wire#powerrail
      { S7_Templates := "SrcType := DInt" } EQ_Contact(in1 := "Unit1.Em2.ControlNodes".SemiAutuSplice.sequence.status.currentStep, in2 := #JOB_5_STEP_01)
      Contact( "Unit1.Em2.ControlNodes".SemiAutuSplice.sequence.status.seqActive )
      wire#w1
      I_Contact( "Unit1.Em2.ControlNodes".cmSplicingLeftModuleMoverFwdBwd.monitoring.inWorkPos )
      wire#w2
      Coil( "Unit1.Em2.ControlNodes".SemiAutuSplice."step".action[501] )
   END_RUNG
   RUNG wire#w1
      I_Contact( "Unit1.Em2.ControlNodes".cmSplicingRightModuleMoverFwdBwd.monitoring.inWorkPos )
   END_RUNG wire#w2
   RUNG wire#w1
      Contact( "Unit1.Em2.ControlNodes".cmSplicingLeftModuleMoverFwdBwd.monitoring.inWorkPos )
      Contact( "Unit1.Em2.ControlNodes".cmSplicingRightModuleMoverFwdBwd.monitoring.inWorkPos )
      Coil( "Unit1.Em2.ControlNodes".SemiAutuSplice."step".transition[501] )
   END_RUNG
   RUNG wire#w1
      Contact( "Unit1.Em2.ControlNodes".SemiAutuSplice."step".transition[501] )
      { S7_Templates := "time_type := Time" } #statTonTimer[501].TON(pt := #SeqDelayTime, et =>)
      Move(in := #STEP_IDLE, out1 => "Unit1.Em2.ControlNodes".SemiAutuSplice.sequence.status.nextStep)
   END_RUNG
   // the same network as SCL:
   #_w1 := ("Unit1.Em2.ControlNodes".SemiAutuSplice.sequence.status.currentStep = #JOB_5_STEP_01) AND "Unit1.Em2.ControlNodes".SemiAutuSplice.sequence.status.seqActive;
   "Unit1.Em2.ControlNodes".SemiAutuSplice."step".action[501] := #_w1 AND (NOT "Unit1.Em2.ControlNodes".cmSplicingLeftModuleMoverFwdBwd.monitoring.inWorkPos OR NOT "Unit1.Em2.ControlNodes".cmSplicingRightModuleMoverFwdBwd.monitoring.inWorkPos);
   "Unit1.Em2.ControlNodes".SemiAutuSplice."step".transition[501] := #_w1 AND "Unit1.Em2.ControlNodes".cmSplicingLeftModuleMoverFwdBwd.monitoring.inWorkPos AND "Unit1.Em2.ControlNodes".cmSplicingRightModuleMoverFwdBwd.monitoring.inWorkPos;
   #statTonTimer[501].TON(IN := #_w1 AND "Unit1.Em2.ControlNodes".SemiAutuSplice."step".transition[501],
                          PT := #SeqDelayTime);
   IF #statTonTimer[501].Q THEN
       "Unit1.Em2.ControlNodes".SemiAutuSplice.sequence.status.nextStep := #STEP_IDLE;
   END_IF;
END_REGION

REGION Network 34: ******************** JOB[7] ELECTRODE VACUUM AUTO ********************
END_REGION

REGION Network 35: Step[701] : Stopper WorkPos Command
   RUNG wire#powerrail
      { S7_Templates := "SrcType := DInt" } EQ_Contact(in1 := "Unit1.Em2.ControlNodes".SemiAutuSplice.sequence.status.currentStep, in2 := #JOB_7_STEP_01)
      Contact( "Unit1.Em2.ControlNodes".SemiAutuSplice.sequence.status.seqActive )
      wire#w1
      I_Contact( "Unit1.Em2.ControlNodes".cmStopperFwdBwd.monitoring.inWorkPos )
      Coil( "Unit1.Em2.ControlNodes".SemiAutuSplice."step".action[701] )
   END_RUNG
   RUNG wire#w1
      Contact( "Unit1.Em2.ControlNodes".cmStopperFwdBwd.monitoring.inWorkPos )
      Coil( "Unit1.Em2.ControlNodes".SemiAutuSplice."step".transition[701] )
   END_RUNG
   RUNG wire#w1
      Contact( "Unit1.Em2.ControlNodes".SemiAutuSplice."step".transition[701] )
      { S7_Templates := "time_type := Time" } #statTonTimer[701].TON(pt := #SeqDelayTime, et =>)
      Move(in := #JOB_7_STEP_11, out1 => "Unit1.Em2.ControlNodes".SemiAutuSplice.sequence.status.nextStep)
   END_RUNG
   // the same network as SCL:
   #_w1 := ("Unit1.Em2.ControlNodes".SemiAutuSplice.sequence.status.currentStep = #JOB_7_STEP_01) AND "Unit1.Em2.ControlNodes".SemiAutuSplice.sequence.status.seqActive;
   "Unit1.Em2.ControlNodes".SemiAutuSplice."step".action[701] := #_w1 AND NOT "Unit1.Em2.ControlNodes".cmStopperFwdBwd.monitoring.inWorkPos;
   "Unit1.Em2.ControlNodes".SemiAutuSplice."step".transition[701] := #_w1 AND "Unit1.Em2.ControlNodes".cmStopperFwdBwd.monitoring.inWorkPos;
   #statTonTimer[701].TON(IN := #_w1 AND "Unit1.Em2.ControlNodes".SemiAutuSplice."step".transition[701],
                          PT := #SeqDelayTime);
   IF #statTonTimer[701].Q THEN
       "Unit1.Em2.ControlNodes".SemiAutuSplice.sequence.status.nextStep := #JOB_7_STEP_11;
   END_IF;
END_REGION

REGION Network 36: Step[711] : Electrode Fix Left Top Down & Electrode Fix Left Bottom Up WorkPos Command
   RUNG wire#powerrail
      { S7_Templates := "SrcType := DInt" } EQ_Contact(in1 := "Unit1.Em2.ControlNodes".SemiAutuSplice.sequence.status.currentStep, in2 := #JOB_7_STEP_11)
      Contact( "Unit1.Em2.ControlNodes".SemiAutuSplice.sequence.status.seqActive )
      wire#w1
      I_Contact( "Unit1.Em2.ControlNodes".cmElectrodeFixLeftTopUpDown.monitoring.inWorkPos )
      wire#w2
      Coil( "Unit1.Em2.ControlNodes".SemiAutuSplice."step".action[711] )
   END_RUNG
   RUNG wire#w1
      I_Contact( "Unit1.Em2.ControlNodes".cmElectrodeFixLeftBottomUpDown.monitoring.inWorkPos )
   END_RUNG wire#w2
   RUNG wire#w1
      Contact( "Unit1.Em2.ControlNodes".cmElectrodeFixLeftTopUpDown.monitoring.inWorkPos )
      Contact( "Unit1.Em2.ControlNodes".cmElectrodeFixLeftBottomUpDown.monitoring.inWorkPos )
      Coil( "Unit1.Em2.ControlNodes".SemiAutuSplice."step".transition[711] )
   END_RUNG
   RUNG wire#w1
      Contact( "Unit1.Em2.ControlNodes".SemiAutuSplice."step".transition[711] )
      { S7_Templates := "time_type := Time" } #statTonTimer[711].TON(pt := #SeqDelayTime, et =>)
      Move(in := #JOB_7_STEP_21, out1 => "Unit1.Em2.ControlNodes".SemiAutuSplice.sequence.status.nextStep)
   END_RUNG
   // the same network as SCL:
   #_w1 := ("Unit1.Em2.ControlNodes".SemiAutuSplice.sequence.status.currentStep = #JOB_7_STEP_11) AND "Unit1.Em2.ControlNodes".SemiAutuSplice.sequence.status.seqActive;
   "Unit1.Em2.ControlNodes".SemiAutuSplice."step".action[711] := #_w1 AND (NOT "Unit1.Em2.ControlNodes".cmElectrodeFixLeftTopUpDown.monitoring.inWorkPos OR NOT "Unit1.Em2.ControlNodes".cmElectrodeFixLeftBottomUpDown.monitoring.inWorkPos);
   "Unit1.Em2.ControlNodes".SemiAutuSplice."step".transition[711] := #_w1 AND "Unit1.Em2.ControlNodes".cmElectrodeFixLeftTopUpDown.monitoring.inWorkPos AND "Unit1.Em2.ControlNodes".cmElectrodeFixLeftBottomUpDown.monitoring.inWorkPos;
   #statTonTimer[711].TON(IN := #_w1 AND "Unit1.Em2.ControlNodes".SemiAutuSplice."step".transition[711],
                          PT := #SeqDelayTime);
   IF #statTonTimer[711].Q THEN
       "Unit1.Em2.ControlNodes".SemiAutuSplice.sequence.status.nextStep := #JOB_7_STEP_21;
   END_IF;
END_REGION

REGION Network 37: Step[721] : Electrode Fix ALL WorkPos Command
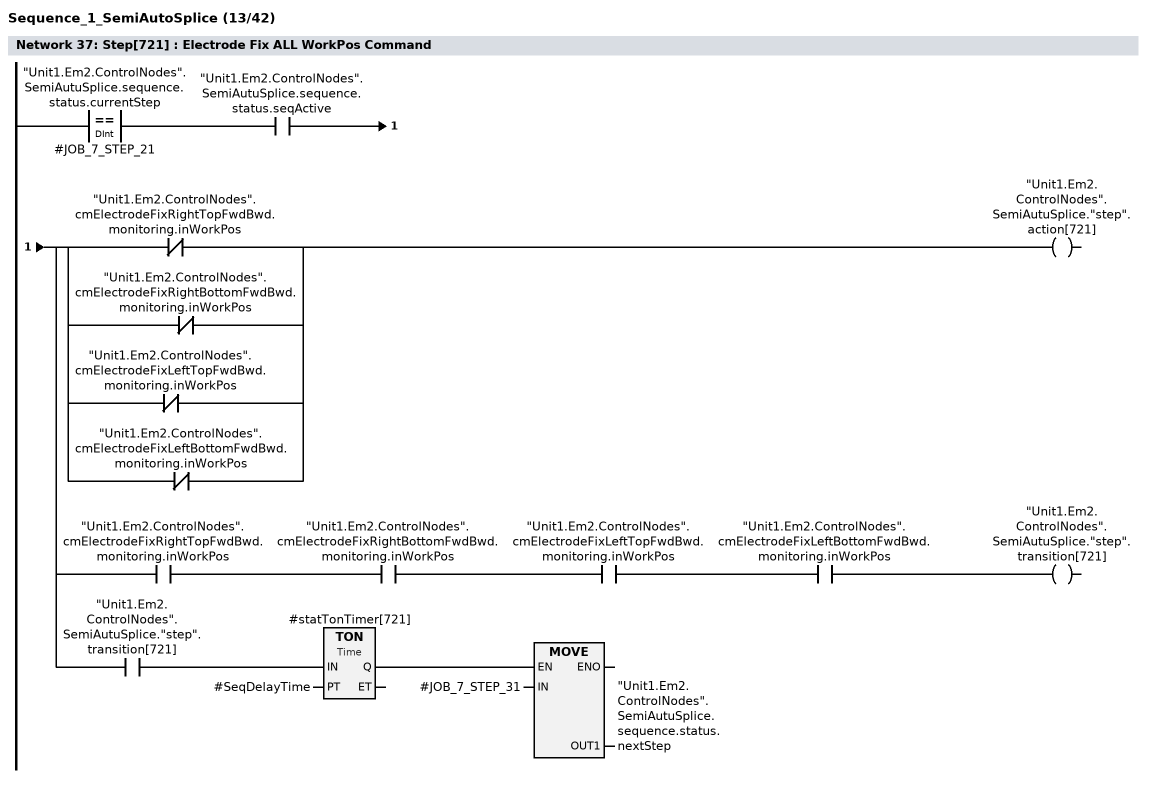
   RUNG wire#powerrail
      { S7_Templates := "SrcType := DInt" } EQ_Contact(in1 := "Unit1.Em2.ControlNodes".SemiAutuSplice.sequence.status.currentStep, in2 := #JOB_7_STEP_21)
      Contact( "Unit1.Em2.ControlNodes".SemiAutuSplice.sequence.status.seqActive )
      wire#w1
      I_Contact( "Unit1.Em2.ControlNodes".cmElectrodeFixRightTopFwdBwd.monitoring.inWorkPos )
      wire#w2
      Coil( "Unit1.Em2.ControlNodes".SemiAutuSplice."step".action[721] )
   END_RUNG
   RUNG wire#w1
      I_Contact( "Unit1.Em2.ControlNodes".cmElectrodeFixRightBottomFwdBwd.monitoring.inWorkPos )
   END_RUNG wire#w2
   RUNG wire#w1
      I_Contact( "Unit1.Em2.ControlNodes".cmElectrodeFixLeftTopFwdBwd.monitoring.inWorkPos )
   END_RUNG wire#w2
   RUNG wire#w1
      I_Contact( "Unit1.Em2.ControlNodes".cmElectrodeFixLeftBottomFwdBwd.monitoring.inWorkPos )
   END_RUNG wire#w2
   RUNG wire#w1
      Contact( "Unit1.Em2.ControlNodes".cmElectrodeFixRightTopFwdBwd.monitoring.inWorkPos )
      Contact( "Unit1.Em2.ControlNodes".cmElectrodeFixRightBottomFwdBwd.monitoring.inWorkPos )
      Contact( "Unit1.Em2.ControlNodes".cmElectrodeFixLeftTopFwdBwd.monitoring.inWorkPos )
      Contact( "Unit1.Em2.ControlNodes".cmElectrodeFixLeftBottomFwdBwd.monitoring.inWorkPos )
      Coil( "Unit1.Em2.ControlNodes".SemiAutuSplice."step".transition[721] )
   END_RUNG
   RUNG wire#w1
      Contact( "Unit1.Em2.ControlNodes".SemiAutuSplice."step".transition[721] )
      { S7_Templates := "time_type := Time" } #statTonTimer[721].TON(pt := #SeqDelayTime, et =>)
      Move(in := #JOB_7_STEP_31, out1 => "Unit1.Em2.ControlNodes".SemiAutuSplice.sequence.status.nextStep)
   END_RUNG
   // the same network as SCL:
   #_w1 := ("Unit1.Em2.ControlNodes".SemiAutuSplice.sequence.status.currentStep = #JOB_7_STEP_21) AND "Unit1.Em2.ControlNodes".SemiAutuSplice.sequence.status.seqActive;
   "Unit1.Em2.ControlNodes".SemiAutuSplice."step".action[721] := #_w1 AND (NOT "Unit1.Em2.ControlNodes".cmElectrodeFixRightTopFwdBwd.monitoring.inWorkPos OR NOT "Unit1.Em2.ControlNodes".cmElectrodeFixRightBottomFwdBwd.monitoring.inWorkPos OR NOT "Unit1.Em2.ControlNodes".cmElectrodeFixLeftTopFwdBwd.monitoring.inWorkPos OR NOT "Unit1.Em2.ControlNodes".cmElectrodeFixLeftBottomFwdBwd.monitoring.inWorkPos);
   "Unit1.Em2.ControlNodes".SemiAutuSplice."step".transition[721] := #_w1 AND "Unit1.Em2.ControlNodes".cmElectrodeFixRightTopFwdBwd.monitoring.inWorkPos AND "Unit1.Em2.ControlNodes".cmElectrodeFixRightBottomFwdBwd.monitoring.inWorkPos AND "Unit1.Em2.ControlNodes".cmElectrodeFixLeftTopFwdBwd.monitoring.inWorkPos AND "Unit1.Em2.ControlNodes".cmElectrodeFixLeftBottomFwdBwd.monitoring.inWorkPos;
   #statTonTimer[721].TON(IN := #_w1 AND "Unit1.Em2.ControlNodes".SemiAutuSplice."step".transition[721],
                          PT := #SeqDelayTime);
   IF #statTonTimer[721].Q THEN
       "Unit1.Em2.ControlNodes".SemiAutuSplice.sequence.status.nextStep := #JOB_7_STEP_31;
   END_IF;
END_REGION

REGION Network 38: Step[731] : Uw Semi Splicer Vacuum All WorkPos Command
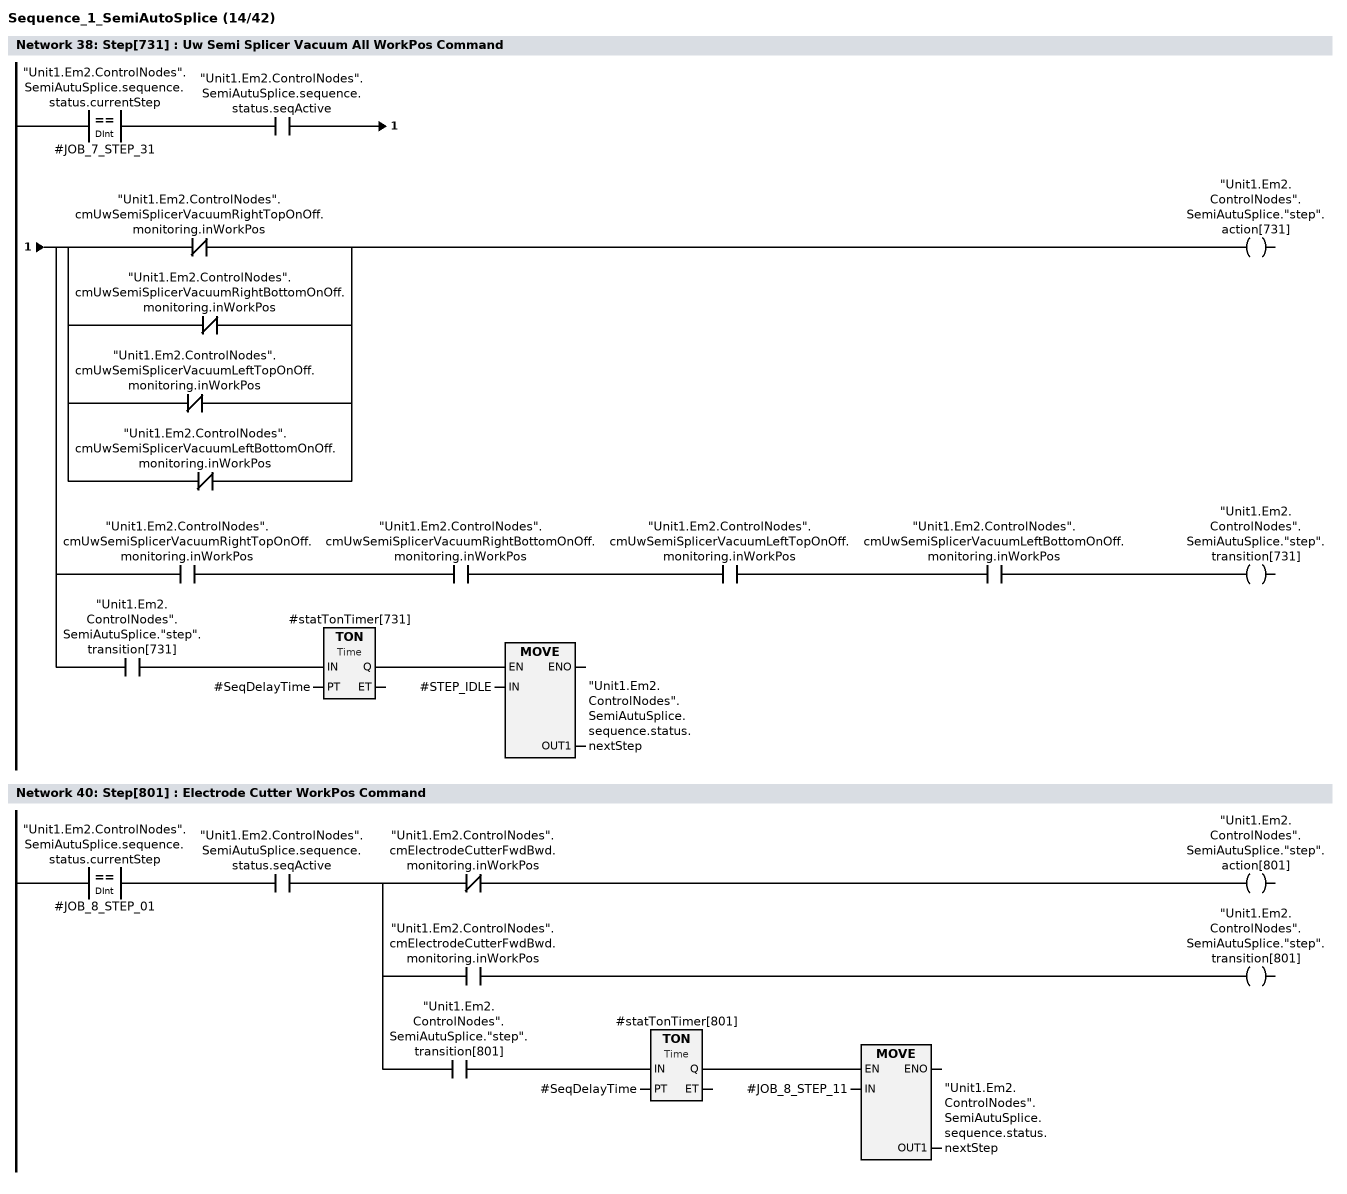
   RUNG wire#powerrail
      { S7_Templates := "SrcType := DInt" } EQ_Contact(in1 := "Unit1.Em2.ControlNodes".SemiAutuSplice.sequence.status.currentStep, in2 := #JOB_7_STEP_31)
      Contact( "Unit1.Em2.ControlNodes".SemiAutuSplice.sequence.status.seqActive )
      wire#w1
      I_Contact( "Unit1.Em2.ControlNodes".cmUwSemiSplicerVacuumRightTopOnOff.monitoring.inWorkPos )
      wire#w2
      Coil( "Unit1.Em2.ControlNodes".SemiAutuSplice."step".action[731] )
   END_RUNG
   RUNG wire#w1
      I_Contact( "Unit1.Em2.ControlNodes".cmUwSemiSplicerVacuumRightBottomOnOff.monitoring.inWorkPos )
   END_RUNG wire#w2
   RUNG wire#w1
      I_Contact( "Unit1.Em2.ControlNodes".cmUwSemiSplicerVacuumLeftTopOnOff.monitoring.inWorkPos )
   END_RUNG wire#w2
   RUNG wire#w1
      I_Contact( "Unit1.Em2.ControlNodes".cmUwSemiSplicerVacuumLeftBottomOnOff.monitoring.inWorkPos )
   END_RUNG wire#w2
   RUNG wire#w1
      Contact( "Unit1.Em2.ControlNodes".cmUwSemiSplicerVacuumRightTopOnOff.monitoring.inWorkPos )
      Contact( "Unit1.Em2.ControlNodes".cmUwSemiSplicerVacuumRightBottomOnOff.monitoring.inWorkPos )
      Contact( "Unit1.Em2.ControlNodes".cmUwSemiSplicerVacuumLeftTopOnOff.monitoring.inWorkPos )
      Contact( "Unit1.Em2.ControlNodes".cmUwSemiSplicerVacuumLeftBottomOnOff.monitoring.inWorkPos )
      Coil( "Unit1.Em2.ControlNodes".SemiAutuSplice."step".transition[731] )
   END_RUNG
   RUNG wire#w1
      Contact( "Unit1.Em2.ControlNodes".SemiAutuSplice."step".transition[731] )
      { S7_Templates := "time_type := Time" } #statTonTimer[731].TON(pt := #SeqDelayTime, et =>)
      Move(in := #STEP_IDLE, out1 => "Unit1.Em2.ControlNodes".SemiAutuSplice.sequence.status.nextStep)
   END_RUNG
   // the same network as SCL:
   #_w1 := ("Unit1.Em2.ControlNodes".SemiAutuSplice.sequence.status.currentStep = #JOB_7_STEP_31) AND "Unit1.Em2.ControlNodes".SemiAutuSplice.sequence.status.seqActive;
   "Unit1.Em2.ControlNodes".SemiAutuSplice."step".action[731] := #_w1 AND (NOT "Unit1.Em2.ControlNodes".cmUwSemiSplicerVacuumRightTopOnOff.monitoring.inWorkPos OR NOT "Unit1.Em2.ControlNodes".cmUwSemiSplicerVacuumRightBottomOnOff.monitoring.inWorkPos OR NOT "Unit1.Em2.ControlNodes".cmUwSemiSplicerVacuumLeftTopOnOff.monitoring.inWorkPos OR NOT "Unit1.Em2.ControlNodes".cmUwSemiSplicerVacuumLeftBottomOnOff.monitoring.inWorkPos);
   "Unit1.Em2.ControlNodes".SemiAutuSplice."step".transition[731] := #_w1 AND "Unit1.Em2.ControlNodes".cmUwSemiSplicerVacuumRightTopOnOff.monitoring.inWorkPos AND "Unit1.Em2.ControlNodes".cmUwSemiSplicerVacuumRightBottomOnOff.monitoring.inWorkPos AND "Unit1.Em2.ControlNodes".cmUwSemiSplicerVacuumLeftTopOnOff.monitoring.inWorkPos AND "Unit1.Em2.ControlNodes".cmUwSemiSplicerVacuumLeftBottomOnOff.monitoring.inWorkPos;
   #statTonTimer[731].TON(IN := #_w1 AND "Unit1.Em2.ControlNodes".SemiAutuSplice."step".transition[731],
                          PT := #SeqDelayTime);
   IF #statTonTimer[731].Q THEN
       "Unit1.Em2.ControlNodes".SemiAutuSplice.sequence.status.nextStep := #STEP_IDLE;
   END_IF;
END_REGION

REGION Network 39: ******************** JOB[8] ELECTRODE CUTTER AUTO ********************
END_REGION

REGION Network 40: Step[801] : Electrode Cutter WorkPos Command
   RUNG wire#powerrail
      { S7_Templates := "SrcType := DInt" } EQ_Contact(in1 := "Unit1.Em2.ControlNodes".SemiAutuSplice.sequence.status.currentStep, in2 := #JOB_8_STEP_01)
      Contact( "Unit1.Em2.ControlNodes".SemiAutuSplice.sequence.status.seqActive )
      wire#w1
      I_Contact( "Unit1.Em2.ControlNodes".cmElectrodeCutterFwdBwd.monitoring.inWorkPos )
      Coil( "Unit1.Em2.ControlNodes".SemiAutuSplice."step".action[801] )
   END_RUNG
   RUNG wire#w1
      Contact( "Unit1.Em2.ControlNodes".cmElectrodeCutterFwdBwd.monitoring.inWorkPos )
      Coil( "Unit1.Em2.ControlNodes".SemiAutuSplice."step".transition[801] )
   END_RUNG
   RUNG wire#w1
      Contact( "Unit1.Em2.ControlNodes".SemiAutuSplice."step".transition[801] )
      { S7_Templates := "time_type := Time" } #statTonTimer[801].TON(pt := #SeqDelayTime, et =>)
      Move(in := #JOB_8_STEP_11, out1 => "Unit1.Em2.ControlNodes".SemiAutuSplice.sequence.status.nextStep)
   END_RUNG
   // the same network as SCL:
   #_w1 := ("Unit1.Em2.ControlNodes".SemiAutuSplice.sequence.status.currentStep = #JOB_8_STEP_01) AND "Unit1.Em2.ControlNodes".SemiAutuSplice.sequence.status.seqActive;
   "Unit1.Em2.ControlNodes".SemiAutuSplice."step".action[801] := #_w1 AND NOT "Unit1.Em2.ControlNodes".cmElectrodeCutterFwdBwd.monitoring.inWorkPos;
   "Unit1.Em2.ControlNodes".SemiAutuSplice."step".transition[801] := #_w1 AND "Unit1.Em2.ControlNodes".cmElectrodeCutterFwdBwd.monitoring.inWorkPos;
   #statTonTimer[801].TON(IN := #_w1 AND "Unit1.Em2.ControlNodes".SemiAutuSplice."step".transition[801],
                          PT := #SeqDelayTime);
   IF #statTonTimer[801].Q THEN
       "Unit1.Em2.ControlNodes".SemiAutuSplice.sequence.status.nextStep := #JOB_8_STEP_11;
   END_IF;
END_REGION

REGION Network 41: Step[811] : Electrode Cutter HomePos Command
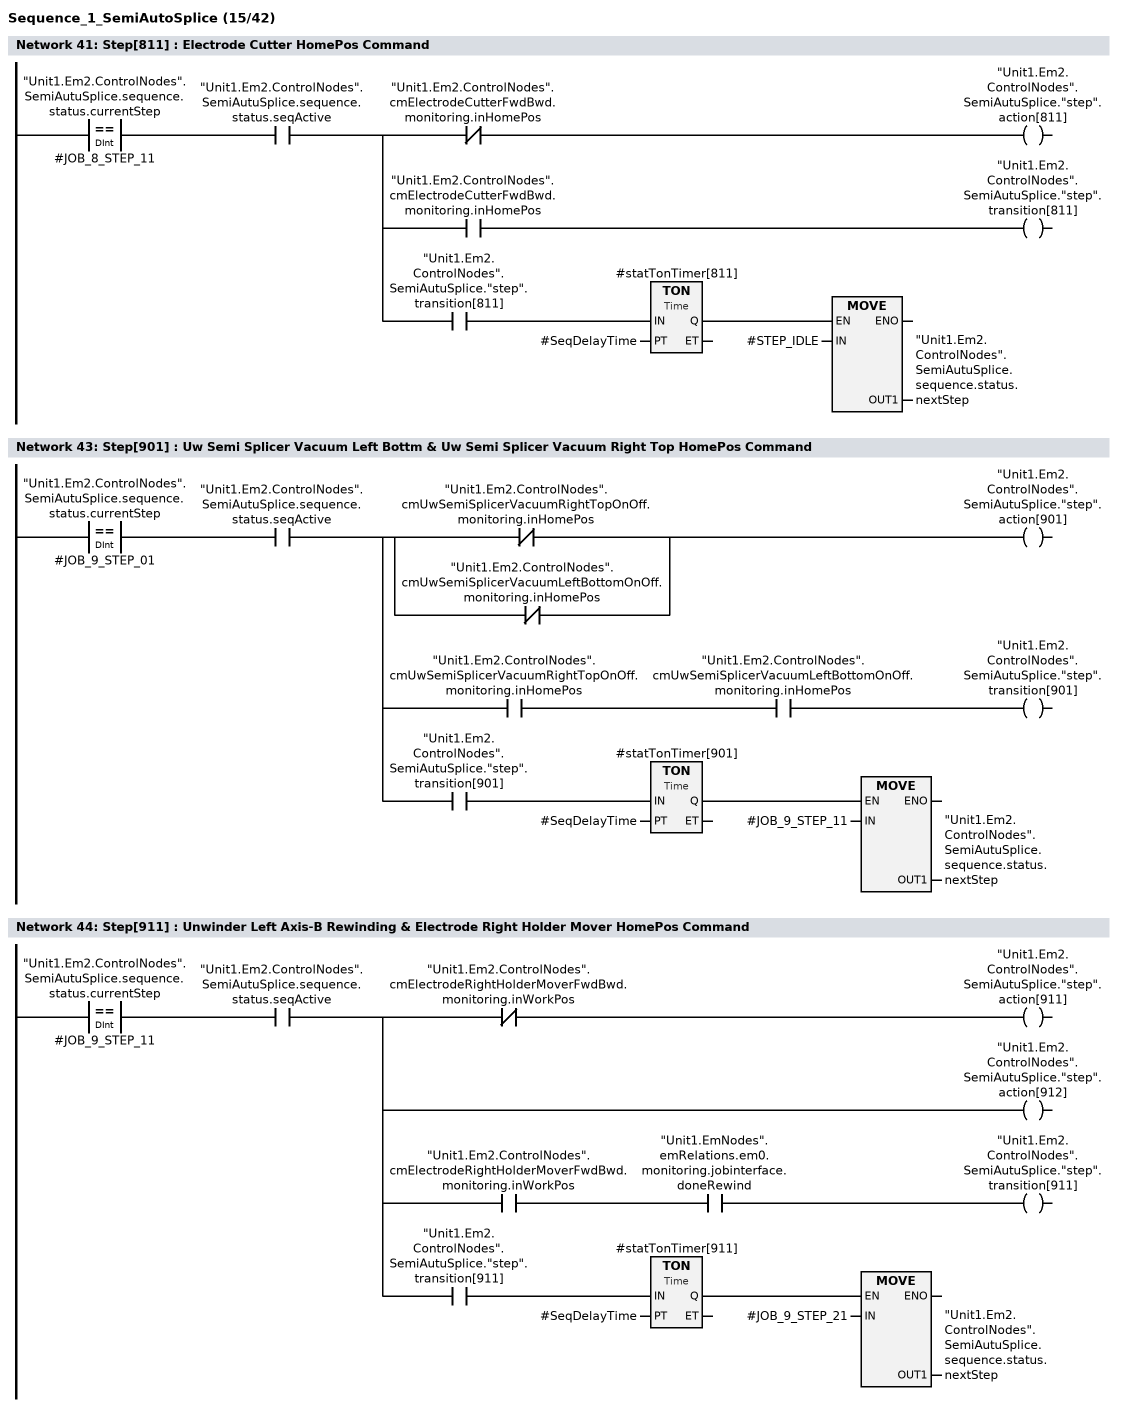
   RUNG wire#powerrail
      { S7_Templates := "SrcType := DInt" } EQ_Contact(in1 := "Unit1.Em2.ControlNodes".SemiAutuSplice.sequence.status.currentStep, in2 := #JOB_8_STEP_11)
      Contact( "Unit1.Em2.ControlNodes".SemiAutuSplice.sequence.status.seqActive )
      wire#w1
      I_Contact( "Unit1.Em2.ControlNodes".cmElectrodeCutterFwdBwd.monitoring.inHomePos )
      Coil( "Unit1.Em2.ControlNodes".SemiAutuSplice."step".action[811] )
   END_RUNG
   RUNG wire#w1
      Contact( "Unit1.Em2.ControlNodes".cmElectrodeCutterFwdBwd.monitoring.inHomePos )
      Coil( "Unit1.Em2.ControlNodes".SemiAutuSplice."step".transition[811] )
   END_RUNG
   RUNG wire#w1
      Contact( "Unit1.Em2.ControlNodes".SemiAutuSplice."step".transition[811] )
      { S7_Templates := "time_type := Time" } #statTonTimer[811].TON(pt := #SeqDelayTime, et =>)
      Move(in := #STEP_IDLE, out1 => "Unit1.Em2.ControlNodes".SemiAutuSplice.sequence.status.nextStep)
   END_RUNG
   // the same network as SCL:
   #_w1 := ("Unit1.Em2.ControlNodes".SemiAutuSplice.sequence.status.currentStep = #JOB_8_STEP_11) AND "Unit1.Em2.ControlNodes".SemiAutuSplice.sequence.status.seqActive;
   "Unit1.Em2.ControlNodes".SemiAutuSplice."step".action[811] := #_w1 AND NOT "Unit1.Em2.ControlNodes".cmElectrodeCutterFwdBwd.monitoring.inHomePos;
   "Unit1.Em2.ControlNodes".SemiAutuSplice."step".transition[811] := #_w1 AND "Unit1.Em2.ControlNodes".cmElectrodeCutterFwdBwd.monitoring.inHomePos;
   #statTonTimer[811].TON(IN := #_w1 AND "Unit1.Em2.ControlNodes".SemiAutuSplice."step".transition[811],
                          PT := #SeqDelayTime);
   IF #statTonTimer[811].Q THEN
       "Unit1.Em2.ControlNodes".SemiAutuSplice.sequence.status.nextStep := #STEP_IDLE;
   END_IF;
END_REGION

REGION Network 42: ******************** JOB[9] LEFT ELECTRODE REMOVER AUTO ********************
END_REGION

REGION Network 43: Step[901] : Uw Semi Splicer Vacuum Left Bottm & Uw Semi Splicer Vacuum Right Top HomePos Command
   RUNG wire#powerrail
      { S7_Templates := "SrcType := DInt" } EQ_Contact(in1 := "Unit1.Em2.ControlNodes".SemiAutuSplice.sequence.status.currentStep, in2 := #JOB_9_STEP_01)
      Contact( "Unit1.Em2.ControlNodes".SemiAutuSplice.sequence.status.seqActive )
      wire#w1
      I_Contact( "Unit1.Em2.ControlNodes".cmUwSemiSplicerVacuumRightTopOnOff.monitoring.inHomePos )
      wire#w2
      Coil( "Unit1.Em2.ControlNodes".SemiAutuSplice."step".action[901] )
   END_RUNG
   RUNG wire#w1
      I_Contact( "Unit1.Em2.ControlNodes".cmUwSemiSplicerVacuumLeftBottomOnOff.monitoring.inHomePos )
   END_RUNG wire#w2
   RUNG wire#w1
      Contact( "Unit1.Em2.ControlNodes".cmUwSemiSplicerVacuumRightTopOnOff.monitoring.inHomePos )
      Contact( "Unit1.Em2.ControlNodes".cmUwSemiSplicerVacuumLeftBottomOnOff.monitoring.inHomePos )
      Coil( "Unit1.Em2.ControlNodes".SemiAutuSplice."step".transition[901] )
   END_RUNG
   RUNG wire#w1
      Contact( "Unit1.Em2.ControlNodes".SemiAutuSplice."step".transition[901] )
      { S7_Templates := "time_type := Time" } #statTonTimer[901].TON(pt := #SeqDelayTime, et =>)
      Move(in := #JOB_9_STEP_11, out1 => "Unit1.Em2.ControlNodes".SemiAutuSplice.sequence.status.nextStep)
   END_RUNG
   // the same network as SCL:
   #_w1 := ("Unit1.Em2.ControlNodes".SemiAutuSplice.sequence.status.currentStep = #JOB_9_STEP_01) AND "Unit1.Em2.ControlNodes".SemiAutuSplice.sequence.status.seqActive;
   "Unit1.Em2.ControlNodes".SemiAutuSplice."step".action[901] := #_w1 AND (NOT "Unit1.Em2.ControlNodes".cmUwSemiSplicerVacuumRightTopOnOff.monitoring.inHomePos OR NOT "Unit1.Em2.ControlNodes".cmUwSemiSplicerVacuumLeftBottomOnOff.monitoring.inHomePos);
   "Unit1.Em2.ControlNodes".SemiAutuSplice."step".transition[901] := #_w1 AND "Unit1.Em2.ControlNodes".cmUwSemiSplicerVacuumRightTopOnOff.monitoring.inHomePos AND "Unit1.Em2.ControlNodes".cmUwSemiSplicerVacuumLeftBottomOnOff.monitoring.inHomePos;
   #statTonTimer[901].TON(IN := #_w1 AND "Unit1.Em2.ControlNodes".SemiAutuSplice."step".transition[901],
                          PT := #SeqDelayTime);
   IF #statTonTimer[901].Q THEN
       "Unit1.Em2.ControlNodes".SemiAutuSplice.sequence.status.nextStep := #JOB_9_STEP_11;
   END_IF;
END_REGION

REGION Network 44: Step[911] : Unwinder Left Axis-B Rewinding & Electrode Right Holder Mover HomePos Command
   RUNG wire#powerrail
      { S7_Templates := "SrcType := DInt" } EQ_Contact(in1 := "Unit1.Em2.ControlNodes".SemiAutuSplice.sequence.status.currentStep, in2 := #JOB_9_STEP_11)
      Contact( "Unit1.Em2.ControlNodes".SemiAutuSplice.sequence.status.seqActive )
      wire#w1
      I_Contact( "Unit1.Em2.ControlNodes".cmElectrodeRightHolderMoverFwdBwd.monitoring.inWorkPos )
      Coil( "Unit1.Em2.ControlNodes".SemiAutuSplice."step".action[911] )
   END_RUNG
   RUNG wire#w1
      Coil( "Unit1.Em2.ControlNodes".SemiAutuSplice."step".action[912] )
   END_RUNG
   RUNG wire#w1
      Contact( "Unit1.Em2.ControlNodes".cmElectrodeRightHolderMoverFwdBwd.monitoring.inWorkPos )
      Contact( "Unit1.EmNodes".emRelations.em0.monitoring.jobinterface.doneRewind )
      Coil( "Unit1.Em2.ControlNodes".SemiAutuSplice."step".transition[911] )
   END_RUNG
   RUNG wire#w1
      Contact( "Unit1.Em2.ControlNodes".SemiAutuSplice."step".transition[911] )
      { S7_Templates := "time_type := Time" } #statTonTimer[911].TON(pt := #SeqDelayTime, et =>)
      Move(in := #JOB_9_STEP_21, out1 => "Unit1.Em2.ControlNodes".SemiAutuSplice.sequence.status.nextStep)
   END_RUNG
   // the same network as SCL:
   #_w1 := ("Unit1.Em2.ControlNodes".SemiAutuSplice.sequence.status.currentStep = #JOB_9_STEP_11) AND "Unit1.Em2.ControlNodes".SemiAutuSplice.sequence.status.seqActive;
   "Unit1.Em2.ControlNodes".SemiAutuSplice."step".action[911] := #_w1 AND NOT "Unit1.Em2.ControlNodes".cmElectrodeRightHolderMoverFwdBwd.monitoring.inWorkPos;
   "Unit1.Em2.ControlNodes".SemiAutuSplice."step".action[912] := #_w1;
   "Unit1.Em2.ControlNodes".SemiAutuSplice."step".transition[911] := #_w1 AND "Unit1.Em2.ControlNodes".cmElectrodeRightHolderMoverFwdBwd.monitoring.inWorkPos AND "Unit1.EmNodes".emRelations.em0.monitoring.jobinterface.doneRewind;
   #statTonTimer[911].TON(IN := #_w1 AND "Unit1.Em2.ControlNodes".SemiAutuSplice."step".transition[911],
                          PT := #SeqDelayTime);
   IF #statTonTimer[911].Q THEN
       "Unit1.Em2.ControlNodes".SemiAutuSplice.sequence.status.nextStep := #JOB_9_STEP_21;
   END_IF;
END_REGION

REGION Network 45: Step[921] : Uw Semi Splicer Vacuum Left Top HomePos & Right Top WorkPos Command
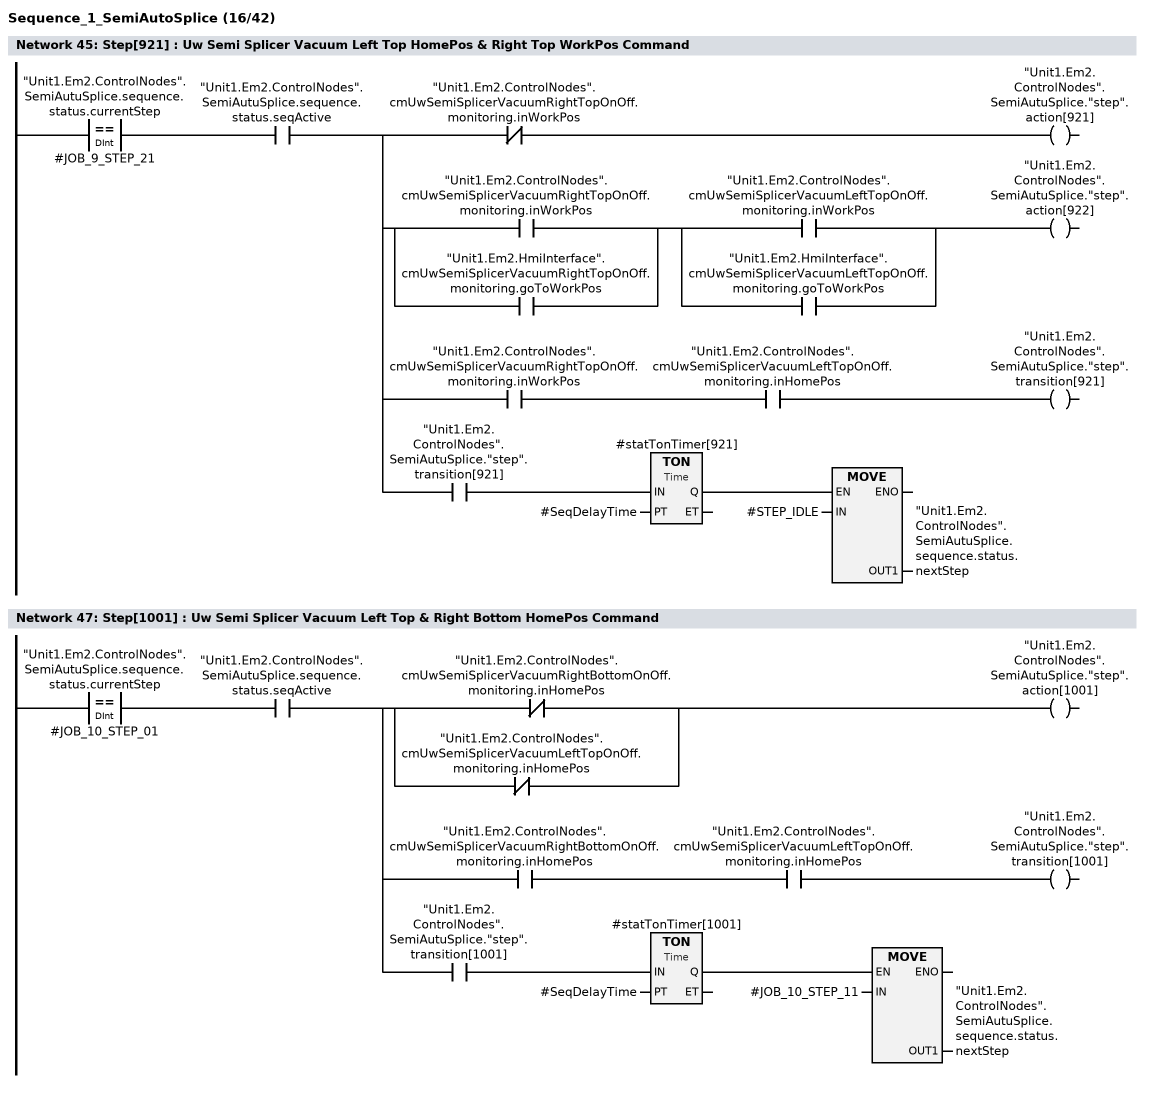
   RUNG wire#powerrail
      { S7_Templates := "SrcType := DInt" } EQ_Contact(in1 := "Unit1.Em2.ControlNodes".SemiAutuSplice.sequence.status.currentStep, in2 := #JOB_9_STEP_21)
      Contact( "Unit1.Em2.ControlNodes".SemiAutuSplice.sequence.status.seqActive )
      wire#w1
      I_Contact( "Unit1.Em2.ControlNodes".cmUwSemiSplicerVacuumRightTopOnOff.monitoring.inWorkPos )
      Coil( "Unit1.Em2.ControlNodes".SemiAutuSplice."step".action[921] )
   END_RUNG
   RUNG wire#w1
      Contact( "Unit1.Em2.ControlNodes".cmUwSemiSplicerVacuumRightTopOnOff.monitoring.inWorkPos )
      wire#w2
      Contact( "Unit1.Em2.ControlNodes".cmUwSemiSplicerVacuumLeftTopOnOff.monitoring.inWorkPos )
      wire#w3
      Coil( "Unit1.Em2.ControlNodes".SemiAutuSplice."step".action[922] )
   END_RUNG
   RUNG wire#w1
      Contact( "Unit1.Em2.HmiInterface".cmUwSemiSplicerVacuumRightTopOnOff.monitoring.goToWorkPos )
   END_RUNG wire#w2
   RUNG wire#w2
      Contact( "Unit1.Em2.HmiInterface".cmUwSemiSplicerVacuumLeftTopOnOff.monitoring.goToWorkPos )
   END_RUNG wire#w3
   RUNG wire#w1
      Contact( "Unit1.Em2.ControlNodes".cmUwSemiSplicerVacuumRightTopOnOff.monitoring.inWorkPos )
      Contact( "Unit1.Em2.ControlNodes".cmUwSemiSplicerVacuumLeftTopOnOff.monitoring.inHomePos )
      Coil( "Unit1.Em2.ControlNodes".SemiAutuSplice."step".transition[921] )
   END_RUNG
   RUNG wire#w1
      Contact( "Unit1.Em2.ControlNodes".SemiAutuSplice."step".transition[921] )
      { S7_Templates := "time_type := Time" } #statTonTimer[921].TON(pt := #SeqDelayTime, et =>)
      Move(in := #STEP_IDLE, out1 => "Unit1.Em2.ControlNodes".SemiAutuSplice.sequence.status.nextStep)
   END_RUNG
   // the same network as SCL:
   #_w1 := ("Unit1.Em2.ControlNodes".SemiAutuSplice.sequence.status.currentStep = #JOB_9_STEP_21) AND "Unit1.Em2.ControlNodes".SemiAutuSplice.sequence.status.seqActive;
   "Unit1.Em2.ControlNodes".SemiAutuSplice."step".action[921] := #_w1 AND NOT "Unit1.Em2.ControlNodes".cmUwSemiSplicerVacuumRightTopOnOff.monitoring.inWorkPos;
   "Unit1.Em2.ControlNodes".SemiAutuSplice."step".action[922] := #_w1 AND ("Unit1.Em2.ControlNodes".cmUwSemiSplicerVacuumRightTopOnOff.monitoring.inWorkPos OR "Unit1.Em2.HmiInterface".cmUwSemiSplicerVacuumRightTopOnOff.monitoring.goToWorkPos) AND ("Unit1.Em2.ControlNodes".cmUwSemiSplicerVacuumLeftTopOnOff.monitoring.inWorkPos OR "Unit1.Em2.HmiInterface".cmUwSemiSplicerVacuumLeftTopOnOff.monitoring.goToWorkPos);
   "Unit1.Em2.ControlNodes".SemiAutuSplice."step".transition[921] := #_w1 AND "Unit1.Em2.ControlNodes".cmUwSemiSplicerVacuumRightTopOnOff.monitoring.inWorkPos AND "Unit1.Em2.ControlNodes".cmUwSemiSplicerVacuumLeftTopOnOff.monitoring.inHomePos;
   #statTonTimer[921].TON(IN := #_w1 AND "Unit1.Em2.ControlNodes".SemiAutuSplice."step".transition[921],
                          PT := #SeqDelayTime);
   IF #statTonTimer[921].Q THEN
       "Unit1.Em2.ControlNodes".SemiAutuSplice.sequence.status.nextStep := #STEP_IDLE;
   END_IF;
END_REGION

REGION Network 46: ******************** JOB[10] RIGHT ELECTRODE REMOVER AUTO ********************
END_REGION

REGION Network 47: Step[1001] : Uw Semi Splicer Vacuum Left Top & Right Bottom HomePos Command
   RUNG wire#powerrail
      { S7_Templates := "SrcType := DInt" } EQ_Contact(in1 := "Unit1.Em2.ControlNodes".SemiAutuSplice.sequence.status.currentStep, in2 := #JOB_10_STEP_01)
      Contact( "Unit1.Em2.ControlNodes".SemiAutuSplice.sequence.status.seqActive )
      wire#w1
      I_Contact( "Unit1.Em2.ControlNodes".cmUwSemiSplicerVacuumRightBottomOnOff.monitoring.inHomePos )
      wire#w2
      Coil( "Unit1.Em2.ControlNodes".SemiAutuSplice."step".action[1001] )
   END_RUNG
   RUNG wire#w1
      I_Contact( "Unit1.Em2.ControlNodes".cmUwSemiSplicerVacuumLeftTopOnOff.monitoring.inHomePos )
   END_RUNG wire#w2
   RUNG wire#w1
      Contact( "Unit1.Em2.ControlNodes".cmUwSemiSplicerVacuumRightBottomOnOff.monitoring.inHomePos )
      Contact( "Unit1.Em2.ControlNodes".cmUwSemiSplicerVacuumLeftTopOnOff.monitoring.inHomePos )
      Coil( "Unit1.Em2.ControlNodes".SemiAutuSplice."step".transition[1001] )
   END_RUNG
   RUNG wire#w1
      Contact( "Unit1.Em2.ControlNodes".SemiAutuSplice."step".transition[1001] )
      { S7_Templates := "time_type := Time" } #statTonTimer[1001].TON(pt := #SeqDelayTime, et =>)
      Move(in := #JOB_10_STEP_11, out1 => "Unit1.Em2.ControlNodes".SemiAutuSplice.sequence.status.nextStep)
   END_RUNG
   // the same network as SCL:
   #_w1 := ("Unit1.Em2.ControlNodes".SemiAutuSplice.sequence.status.currentStep = #JOB_10_STEP_01) AND "Unit1.Em2.ControlNodes".SemiAutuSplice.sequence.status.seqActive;
   "Unit1.Em2.ControlNodes".SemiAutuSplice."step".action[1001] := #_w1 AND (NOT "Unit1.Em2.ControlNodes".cmUwSemiSplicerVacuumRightBottomOnOff.monitoring.inHomePos OR NOT "Unit1.Em2.ControlNodes".cmUwSemiSplicerVacuumLeftTopOnOff.monitoring.inHomePos);
   "Unit1.Em2.ControlNodes".SemiAutuSplice."step".transition[1001] := #_w1 AND "Unit1.Em2.ControlNodes".cmUwSemiSplicerVacuumRightBottomOnOff.monitoring.inHomePos AND "Unit1.Em2.ControlNodes".cmUwSemiSplicerVacuumLeftTopOnOff.monitoring.inHomePos;
   #statTonTimer[1001].TON(IN := #_w1 AND "Unit1.Em2.ControlNodes".SemiAutuSplice."step".transition[1001],
                           PT := #SeqDelayTime);
   IF #statTonTimer[1001].Q THEN
       "Unit1.Em2.ControlNodes".SemiAutuSplice.sequence.status.nextStep := #JOB_10_STEP_11;
   END_IF;
END_REGION

REGION Network 48: Step[1011] : Unwinder Right Axis-B Rewinding & Electrode Left Holder Mover HomePos Command
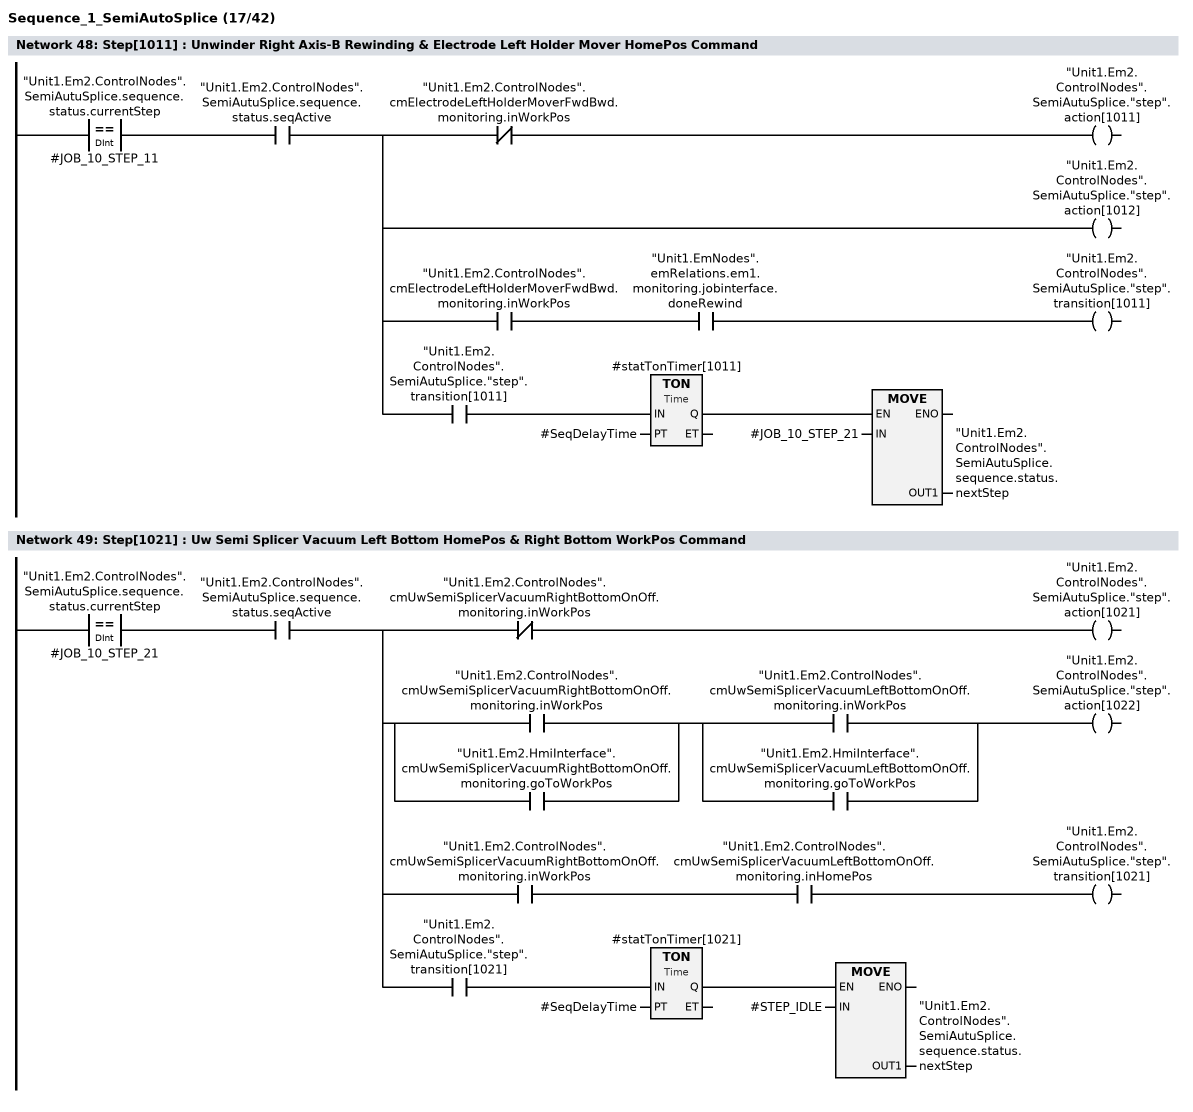
   RUNG wire#powerrail
      { S7_Templates := "SrcType := DInt" } EQ_Contact(in1 := "Unit1.Em2.ControlNodes".SemiAutuSplice.sequence.status.currentStep, in2 := #JOB_10_STEP_11)
      Contact( "Unit1.Em2.ControlNodes".SemiAutuSplice.sequence.status.seqActive )
      wire#w1
      I_Contact( "Unit1.Em2.ControlNodes".cmElectrodeLeftHolderMoverFwdBwd.monitoring.inWorkPos )
      Coil( "Unit1.Em2.ControlNodes".SemiAutuSplice."step".action[1011] )
   END_RUNG
   RUNG wire#w1
      Coil( "Unit1.Em2.ControlNodes".SemiAutuSplice."step".action[1012] )
   END_RUNG
   RUNG wire#w1
      Contact( "Unit1.Em2.ControlNodes".cmElectrodeLeftHolderMoverFwdBwd.monitoring.inWorkPos )
      Contact( "Unit1.EmNodes".emRelations.em1.monitoring.jobinterface.doneRewind )
      Coil( "Unit1.Em2.ControlNodes".SemiAutuSplice."step".transition[1011] )
   END_RUNG
   RUNG wire#w1
      Contact( "Unit1.Em2.ControlNodes".SemiAutuSplice."step".transition[1011] )
      { S7_Templates := "time_type := Time" } #statTonTimer[1011].TON(pt := #SeqDelayTime, et =>)
      Move(in := #JOB_10_STEP_21, out1 => "Unit1.Em2.ControlNodes".SemiAutuSplice.sequence.status.nextStep)
   END_RUNG
   // the same network as SCL:
   #_w1 := ("Unit1.Em2.ControlNodes".SemiAutuSplice.sequence.status.currentStep = #JOB_10_STEP_11) AND "Unit1.Em2.ControlNodes".SemiAutuSplice.sequence.status.seqActive;
   "Unit1.Em2.ControlNodes".SemiAutuSplice."step".action[1011] := #_w1 AND NOT "Unit1.Em2.ControlNodes".cmElectrodeLeftHolderMoverFwdBwd.monitoring.inWorkPos;
   "Unit1.Em2.ControlNodes".SemiAutuSplice."step".action[1012] := #_w1;
   "Unit1.Em2.ControlNodes".SemiAutuSplice."step".transition[1011] := #_w1 AND "Unit1.Em2.ControlNodes".cmElectrodeLeftHolderMoverFwdBwd.monitoring.inWorkPos AND "Unit1.EmNodes".emRelations.em1.monitoring.jobinterface.doneRewind;
   #statTonTimer[1011].TON(IN := #_w1 AND "Unit1.Em2.ControlNodes".SemiAutuSplice."step".transition[1011],
                           PT := #SeqDelayTime);
   IF #statTonTimer[1011].Q THEN
       "Unit1.Em2.ControlNodes".SemiAutuSplice.sequence.status.nextStep := #JOB_10_STEP_21;
   END_IF;
END_REGION

